LIN {X 0,Y 251.586,Z 580.66,A -85,B 0,C 180,E1 17106.896,E2 17106.896} C_VEL
LIN {X 0,Y 250.824,Z 580.66,A -85,B 0,C 180,E1 17115.723,E2 17115.723} C_VEL
LIN {X 0,Y 250.856,Z 581.328,A -85,B 0,C 180,E1 17116.877,E2 17116.877} C_VEL
LIN {X 0,Y 252.882,Z 586.254,A -85,B 0,C 180,E1 17118.487,E2 17118.487} C_VEL
LIN {X 0,Y 255.97,Z 589.116,A -85,B 0,C 180,E1 17120.381,E2 17120.381} C_VEL
LIN {X 0,Y 260.025,Z 594.777,A -85,B 0,C 180,E1 17122.728,E2 17122.728} C_VEL
LIN {X 0,Y 273.524,Z 615.35,A -85,B 0,C 180,E1 17129.206,E2 17129.206} C_VEL
LIN {X 0,Y 285.886,Z 637.872,A -85,B 0,C 180,E1 17134.459,E2 17134.459} C_VEL
LIN {X 0,Y 296.581,Z 664.88,A -85,B 0,C 180,E1 17139.344,E2 17139.344} C_VEL
LIN {X 0,Y 300.476,Z 680.869,A -85,B 0,C 180,E1 17141.812,E2 17141.812} C_VEL
LIN {X 0,Y 290.892,Z 714.694,A -85,B 0,C 180,E1 17144.762,E2 17144.762} C_VEL
LIN {X 0,Y 280.033,Z 747.013,A -85,B 0,C 180,E1 17149.078,E2 17149.078} C_VEL
LIN {X 0,Y 269.468,Z 775.475,A -85,B 0,C 180,E1 17154.67,E2 17154.67} C_VEL
LIN {X 0,Y 261.005,Z 799.602,A -85,B 0,C 180,E1 17161.584,E2 17161.584} C_VEL
LIN {X 0,Y 255.731,Z 817.938,A -85,B 0,C 180,E1 17169.263,E2 17169.263} C_VEL
LIN {X 0,Y 254.018,Z 830.311,A -85,B 0,C 180,E1 17177.144,E2 17177.144} C_VEL
LIN {X 0,Y 254.336,Z 835.933,A -85,B 0,C 180,E1 17183.183,E2 17183.183} C_VEL
LIN {X 0,Y 254.787,Z 838.259,A -85,B 0,C 180,E1 17189.997,E2 17189.997} C_VEL
LIN {X 0,Y 254.301,Z 835.944,A -85,B 0,C 180,E1 17196.813,E2 17196.813} C_VEL
LIN {X 0,Y 254.151,Z 828.084,A -85,B 0,C 180,E1 17204.612,E2 17204.612} C_VEL
LIN {X 0,Y 256.598,Z 814.491,A -85,B 0,C 180,E1 17212.469,E2 17212.469} C_VEL
LIN {X 0,Y 262.523,Z 794.979,A -85,B 0,C 180,E1 17219.974,E2 17219.974} C_VEL
LIN {X 0,Y 271.462,Z 770.337,A -85,B 0,C 180,E1 17226.54,E2 17226.54} C_VEL
LIN {X 0,Y 281.993,Z 741.378,A -85,B 0,C 180,E1 17231.838,E2 17231.838} C_VEL
LIN {X 0,Y 292.893,Z 708.642,A -85,B 0,C 180,E1 17235.888,E2 17235.888} C_VEL
LIN {X 0,Y 300.451,Z 679.152,A -85,B 0,C 180,E1 17238.429,E2 17238.429} C_VEL
LIN {X 0,Y 291.372,Z 650.188,A -85,B 0,C 180,E1 17243.212,E2 17243.212} C_VEL
LIN {X 0,Y 279.017,Z 624.432,A -85,B 0,C 180,E1 17248.514,E2 17248.514} C_VEL
LIN {X 0,Y 264.583,Z 601.351,A -85,B 0,C 180,E1 17255.009,E2 17255.009} C_VEL
LIN {X 0,Y 258.73,Z 593.721,A -85,B 0,C 180,E1 17258.055,E2 17258.055} C_VEL
LIN {X 0,Y 254.701,Z 587.628,A -85,B 0,C 180,E1 17260.528,E2 17260.528} C_VEL
LIN {X 0,Y 251.195,Z 583.366,A -85,B 0,C 180,E1 17262.902,E2 17262.902} C_VEL
LIN {X 0,Y 250.74,Z 580.66,A -85,B 0,C 180,E1 17263.513,E2 17263.513} C_VEL
LIN {X 0,Y 250.771,Z 580.66,A -85,B 0,C 180,E1 17264.591,E2 17264.591} C_VEL
LIN {X 0,Y 248.407,Z 580.66,A -85,B 0,C 180,E1 17267.555,E2 17267.555} C_VEL
LIN {X 0,Y 243.524,Z 580.66,A -85,B 0,C 180,E1 17272.588,E2 17272.588} C_VEL
LIN {X 0,Y 244.313,Z 580.66,A -85,B 0,C 180,E1 17279.993,E2 17279.993} C_VEL
LIN {X 0,Y 243.604,Z 580.66,A -85,B 0,C 180,E1 17287.689,E2 17287.689} C_VEL
LIN {X 0,Y 242.887,Z 581.231,A -85,B 0,C 180,E1 17296.498,E2 17296.498} C_VEL
LIN {X 0,Y 245.095,Z 586.44,A -85,B 0,C 180,E1 17299.111,E2 17299.111} C_VEL
LIN {X 0,Y 248.217,Z 589.119,A -85,B 0,C 180,E1 17301.735,E2 17301.735} C_VEL
LIN {X 0,Y 251.98,Z 594.885,A -85,B 0,C 180,E1 17304.775,E2 17304.775} C_VEL
LIN {X 0,Y 258.821,Z 606.093,A -85,B 0,C 180,E1 17309.635,E2 17309.635} C_VEL
LIN {X 0,Y 266.343,Z 619.396,A -85,B 0,C 180,E1 17314.5,E2 17314.5} C_VEL
LIN {X 0,Y 275.183,Z 640.528,A -85,B 0,C 180,E1 17320.618,E2 17320.618} C_VEL
LIN {X 0,Y 280.604,Z 660.927,A -85,B 0,C 180,E1 17325.778,E2 17325.778} C_VEL
LIN {X 0,Y 283.15,Z 682.748,A -85,B 0,C 180,E1 17331.089,E2 17331.089} C_VEL
LIN {X 0,Y 282.39,Z 690.579,A -85,B 0,C 180,E1 17332.879,E2 17332.879} C_VEL
LIN {X 0,Y 271.737,Z 715.104,A -85,B 0,C 180,E1 17338.165,E2 17338.165} C_VEL
LIN {X 0,Y 262.088,Z 734.388,A -85,B 0,C 180,E1 17344.421,E2 17344.421} C_VEL
LIN {X 0,Y 254.304,Z 749.195,A -85,B 0,C 180,E1 17351.948,E2 17351.948} C_VEL
LIN {X 0,Y 249.965,Z 757.81,A -85,B 0,C 180,E1 17359.569,E2 17359.569} C_VEL
LIN {X 0,Y 248.341,Z 761.384,A -85,B 0,C 180,E1 17366.52,E2 17366.52} C_VEL
LIN {X 0,Y 248.401,Z 761.339,A -85,B 0,C 180,E1 17373.486,E2 17373.486} C_VEL
LIN {X 0,Y 250.691,Z 756.218,A -85,B 0,C 180,E1 17382.164,E2 17382.164} C_VEL
LIN {X 0,Y 256.072,Z 745.785,A -85,B 0,C 180,E1 17390.024,E2 17390.024} C_VEL
LIN {X 0,Y 264.332,Z 729.864,A -85,B 0,C 180,E1 17397.176,E2 17397.176} C_VEL
LIN {X 0,Y 274.613,Z 708.641,A -85,B 0,C 180,E1 17403.334,E2 17403.334} C_VEL
LIN {X 0,Y 283.087,Z 687.119,A -85,B 0,C 180,E1 17407.736,E2 17407.736} C_VEL
LIN {X 0,Y 281.313,Z 665.464,A -85,B 0,C 180,E1 17413.014,E2 17413.014} C_VEL
LIN {X 0,Y 276.056,Z 643.398,A -85,B 0,C 180,E1 17418.477,E2 17418.477} C_VEL
LIN {X 0,Y 268.072,Z 623.359,A -85,B 0,C 180,E1 17424.148,E2 17424.148} C_VEL
LIN {X 0,Y 259.698,Z 607.475,A -85,B 0,C 180,E1 17429.607,E2 17429.607} C_VEL
LIN {X 0,Y 251.831,Z 594.8,A -85,B 0,C 180,E1 17435.08,E2 17435.08} C_VEL
LIN {X 0,Y 248.171,Z 589.103,A -85,B 0,C 180,E1 17438.026,E2 17438.026} C_VEL
LIN {X 0,Y 243.16,Z 583.155,A -85,B 0,C 180,E1 17442.656,E2 17442.656} C_VEL
LIN {X 0,Y 242.76,Z 580.66,A -85,B 0,C 180,E1 17443.348,E2 17443.348} C_VEL
LIN {X 0,Y 243.579,Z 580.66,A -85,B 0,C 180,E1 17452.89,E2 17452.89} C_VEL
LIN {X 0,Y 244.286,Z 580.66,A -85,B 0,C 180,E1 17460.007,E2 17460.007} C_VEL
LIN {X 0,Y 243.579,Z 580.66,A -85,B 0,C 180,E1 17467.599,E2 17467.599} C_VEL
LIN {X 0,Y 243.293,Z 581.322,A -85,B 0,C 180,E1 17471.182,E2 17471.182} C_VEL
LIN {X 0,Y 245.218,Z 586.034,A -85,B 0,C 180,E1 17473.348,E2 17473.348} C_VEL
LIN {X 0,Y 248.738,Z 589.237,A -85,B 0,C 180,E1 17476.195,E2 17476.195} C_VEL
LIN {X 0,Y 252.376,Z 594.794,A -85,B 0,C 180,E1 17478.864,E2 17478.864} C_VEL
LIN {X 0,Y 259.902,Z 605.854,A -85,B 0,C 180,E1 17483.417,E2 17483.417} C_VEL
LIN {X 0,Y 270.347,Z 622.266,A -85,B 0,C 180,E1 17488.668,E2 17488.668} C_VEL
LIN {X 0,Y 281.614,Z 643.967,A -85,B 0,C 180,E1 17493.894,E2 17493.894} C_VEL
LIN {X 0,Y 291.407,Z 670.701,A -85,B 0,C 180,E1 17498.927,E2 17498.927} C_VEL
LIN {X 0,Y 293.962,Z 683.793,A -85,B 0,C 180,E1 17500.965,E2 17500.965} C_VEL
LIN {X 0,Y 283.468,Z 718.719,A -85,B 0,C 180,E1 17504.224,E2 17504.224} C_VEL
LIN {X 0,Y 272.472,Z 749.515,A -85,B 0,C 180,E1 17508.614,E2 17508.614} C_VEL
LIN {X 0,Y 261.648,Z 777.115,A -85,B 0,C 180,E1 17514.349,E2 17514.349} C_VEL
LIN {X 0,Y 253.011,Z 800.517,A -85,B 0,C 180,E1 17521.5,E2 17521.5} C_VEL
LIN {X 0,Y 247.643,Z 818.557,A -85,B 0,C 180,E1 17529.58,E2 17529.58} C_VEL
LIN {X 0,Y 246.171,Z 829.932,A -85,B 0,C 180,E1 17537.467,E2 17537.467} C_VEL
LIN {X 0,Y 246.479,Z 834.73,A -85,B 0,C 180,E1 17542.964,E2 17542.964} C_VEL
LIN {X 0,Y 246.965,Z 837.071,A -85,B 0,C 180,E1 17549.997,E2 17549.997} C_VEL
LIN {X 0,Y 246.446,Z 834.741,A -85,B 0,C 180,E1 17557.031,E2 17557.031} C_VEL
LIN {X 0,Y 246.335,Z 826.853,A -85,B 0,C 180,E1 17565.087,E2 17565.087} C_VEL
LIN {X 0,Y 249.016,Z 813.226,A -85,B 0,C 180,E1 17573.192,E2 17573.192} C_VEL
LIN {X 0,Y 255.521,Z 793.456,A -85,B 0,C 180,E1 17580.975,E2 17580.975} C_VEL
LIN {X 0,Y 265.153,Z 768.4,A -85,B 0,C 180,E1 17587.736,E2 17587.736} C_VEL
LIN {X 0,Y 276.224,Z 739.373,A -85,B 0,C 180,E1 17593.062,E2 17593.062} C_VEL
LIN {X 0,Y 287.3,Z 707.205,A -85,B 0,C 180,E1 17597.048,E2 17597.048} C_VEL
LIN {X 0,Y 294.084,Z 681.567,A -85,B 0,C 180,E1 17599.32,E2 17599.32} C_VEL
LIN {X 0,Y 285.773,Z 653.755,A -85,B 0,C 180,E1 17604.182,E2 17604.182} C_VEL
LIN {X 0,Y 274.795,Z 629.935,A -85,B 0,C 180,E1 17609.355,E2 17609.355} C_VEL
LIN {X 0,Y 261.915,Z 608.278,A -85,B 0,C 180,E1 17615.646,E2 17615.646} C_VEL
LIN {X 0,Y 252.419,Z 594.824,A -85,B 0,C 180,E1 17621.252,E2 17621.252} C_VEL
LIN {X 0,Y 248.765,Z 589.298,A -85,B 0,C 180,E1 17623.95,E2 17623.95} C_VEL
LIN {X 0,Y 243.476,Z 582.895,A -85,B 0,C 180,E1 17628.714,E2 17628.714} C_VEL
LIN {X 0,Y 243.245,Z 580.66,A -85,B 0,C 180,E1 17629.268,E2 17629.268} C_VEL
LIN {X 0,Y 243.524,Z 580.66,A -85,B 0,C 180,E1 17632.588,E2 17632.588} C_VEL
LIN {X 0,Y 241.56,Z 580.866,A -85,B 0,C 180,E1 17635.609,E2 17635.609} C_VEL
LIN {X 0,Y 236.308,Z 581.372,A -85,B 0,C 180,E1 17640.735,E2 17640.735} C_VEL
LIN {X 0,Y 236.125,Z 582.654,A -85,B 0,C 180,E1 17645.034,E2 17645.034} C_VEL
LIN {X 0,Y 241.213,Z 589.227,A -85,B 0,C 180,E1 17655.935,E2 17655.935} C_VEL
LIN {X 0,Y 244.265,Z 594.75,A -85,B 0,C 180,E1 17659.521,E2 17659.521} C_VEL
LIN {X 0,Y 246.174,Z 596.995,A -85,B 0,C 180,E1 17661.317,E2 17661.317} C_VEL
LIN {X 0,Y 251.017,Z 604.941,A -85,B 0,C 180,E1 17665.534,E2 17665.534} C_VEL
LIN {X 0,Y 257.986,Z 617.049,A -85,B 0,C 180,E1 17670.773,E2 17670.773} C_VEL
LIN {X 0,Y 266.924,Z 636.801,A -85,B 0,C 180,E1 17677.416,E2 17677.416} C_VEL
LIN {X 0,Y 273.626,Z 659.052,A -85,B 0,C 180,E1 17683.579,E2 17683.579} C_VEL
LIN {X 0,Y 276.511,Z 682.15,A -85,B 0,C 180,E1 17689.455,E2 17689.455} C_VEL
LIN {X 0,Y 276.319,Z 691.581,A -85,B 0,C 180,E1 17691.853,E2 17691.853} C_VEL
LIN {X 0,Y 265.14,Z 716.323,A -85,B 0,C 180,E1 17697.276,E2 17697.276} C_VEL
LIN {X 0,Y 255.049,Z 735.593,A -85,B 0,C 180,E1 17703.662,E2 17703.662} C_VEL
LIN {X 0,Y 246.833,Z 750.462,A -85,B 0,C 180,E1 17711.439,E2 17711.439} C_VEL
LIN {X 0,Y 242.281,Z 758.998,A -85,B 0,C 180,E1 17719.235,E2 17719.235} C_VEL
LIN {X 0,Y 240.563,Z 762.567,A -85,B 0,C 180,E1 17726.407,E2 17726.407} C_VEL
LIN {X 0,Y 240.61,Z 762.525,A -85,B 0,C 180,E1 17733.599,E2 17733.599} C_VEL
LIN {X 0,Y 242.41,Z 758.874,A -85,B 0,C 180,E1 17740.766,E2 17740.766} C_VEL
LIN {X 0,Y 247.584,Z 749.058,A -85,B 0,C 180,E1 17749.377,E2 17749.377} C_VEL
LIN {X 0,Y 256.295,Z 733.262,A -85,B 0,C 180,E1 17757.15,E2 17757.15} C_VEL
LIN {X 0,Y 266.64,Z 712.908,A -85,B 0,C 180,E1 17763.491,E2 17763.491} C_VEL
LIN {X 0,Y 276.473,Z 689.578,A -85,B 0,C 180,E1 17768.516,E2 17768.516} C_VEL
LIN {X 0,Y 275.106,Z 668.329,A -85,B 0,C 180,E1 17773.924,E2 17773.924} C_VEL
LIN {X 0,Y 270.275,Z 646.652,A -85,B 0,C 180,E1 17779.593,E2 17779.593} C_VEL
LIN {X 0,Y 262.338,Z 625.74,A -85,B 0,C 180,E1 17785.898,E2 17785.898} C_VEL
LIN {X 0,Y 253.002,Z 608.092,A -85,B 0,C 180,E1 17792.719,E2 17792.719} C_VEL
LIN {X 0,Y 248.7,Z 601.295,A -85,B 0,C 180,E1 17796.152,E2 17796.152} C_VEL
LIN {X 0,Y 244.968,Z 595.242,A -85,B 0,C 180,E1 17799.546,E2 17799.546} C_VEL
LIN {X 0,Y 241.374,Z 590.26,A -85,B 0,C 180,E1 17803.368,E2 17803.368} C_VEL
LIN {X 0,Y 240.62,Z 588.252,A -85,B 0,C 180,E1 17804.452,E2 17804.452} C_VEL
LIN {X 0,Y 235.904,Z 581.705,A -85,B 0,C 180,E1 17815.076,E2 17815.076} C_VEL
LIN {X 0,Y 236.078,Z 580.66,A -85,B 0,C 180,E1 17816.342,E2 17816.342} C_VEL
LIN {X 0,Y 236.288,Z 581.54,A -85,B 0,C 180,E1 17820.693,E2 17820.693} C_VEL
LIN {X 0,Y 239.8,Z 587.635,A -85,B 0,C 180,E1 17828.388,E2 17828.388} C_VEL
LIN {X 0,Y 241.633,Z 589.26,A -85,B 0,C 180,E1 17830.576,E2 17830.576} C_VEL
LIN {X 0,Y 244.962,Z 594.756,A -85,B 0,C 180,E1 17834.043,E2 17834.043} C_VEL
LIN {X 0,Y 246.995,Z 597.157,A -85,B 0,C 180,E1 17835.735,E2 17835.735} C_VEL
LIN {X 0,Y 252.731,Z 605.965,A -85,B 0,C 180,E1 17839.97,E2 17839.97} C_VEL
LIN {X 0,Y 260.813,Z 618.329,A -85,B 0,C 180,E1 17844.805,E2 17844.805} C_VEL
LIN {X 0,Y 272.421,Z 639.11,A -85,B 0,C 180,E1 17850.826,E2 17850.826} C_VEL
LIN {X 0,Y 282.893,Z 665.351,A -85,B 0,C 180,E1 17856.451,E2 17856.451} C_VEL
LIN {X 0,Y 287.919,Z 685.239,A -85,B 0,C 180,E1 17859.975,E2 17859.975} C_VEL
LIN {X 0,Y 277.123,Z 719.417,A -85,B 0,C 180,E1 17863.279,E2 17863.279} C_VEL
LIN {X 0,Y 265.896,Z 749.338,A -85,B 0,C 180,E1 17867.649,E2 17867.649} C_VEL
LIN {X 0,Y 254.445,Z 777.14,A -85,B 0,C 180,E1 17873.625,E2 17873.625} C_VEL
LIN {X 0,Y 245.387,Z 800.43,A -85,B 0,C 180,E1 17881.034,E2 17881.034} C_VEL
LIN {X 0,Y 239.746,Z 818.454,A -85,B 0,C 180,E1 17889.597,E2 17889.597} C_VEL
LIN {X 0,Y 238.305,Z 828.85,A -85,B 0,C 180,E1 17897.193,E2 17897.193} C_VEL
LIN {X 0,Y 238.603,Z 833.523,A -85,B 0,C 180,E1 17902.731,E2 17902.731} C_VEL
LIN {X 0,Y 239.168,Z 835.886,A -85,B 0,C 180,E1 17909.997,E2 17909.997} C_VEL
LIN {X 0,Y 238.571,Z 833.536,A -85,B 0,C 180,E1 17917.264,E2 17917.264} C_VEL
LIN {X 0,Y 238.535,Z 825.622,A -85,B 0,C 180,E1 17925.592,E2 17925.592} C_VEL
LIN {X 0,Y 241.516,Z 811.968,A -85,B 0,C 180,E1 17933.957,E2 17933.957} C_VEL
LIN {X 0,Y 248.658,Z 791.721,A -85,B 0,C 180,E1 17942.106,E2 17942.106} C_VEL
LIN {X 0,Y 258.886,Z 766.728,A -85,B 0,C 180,E1 17948.921,E2 17948.921} C_VEL
LIN {X 0,Y 270.352,Z 738.015,A -85,B 0,C 180,E1 17954.236,E2 17954.236} C_VEL
LIN {X 0,Y 282.033,Z 705.186,A -85,B 0,C 180,E1 17958.307,E2 17958.307} C_VEL
LIN {X 0,Y 287.845,Z 684.025,A -85,B 0,C 180,E1 17960.236,E2 17960.236} C_VEL
LIN {X 0,Y 280.608,Z 658.457,A -85,B 0,C 180,E1 17964.931,E2 17964.931} C_VEL
LIN {X 0,Y 270.497,Z 635.303,A -85,B 0,C 180,E1 17970.205,E2 17970.205} C_VEL
LIN {X 0,Y 258.809,Z 614.731,A -85,B 0,C 180,E1 17976.478,E2 17976.478} C_VEL
LIN {X 0,Y 250.138,Z 601.941,A -85,B 0,C 180,E1 17981.985,E2 17981.985} C_VEL
LIN {X 0,Y 245.7,Z 595.309,A -85,B 0,C 180,E1 17985.546,E2 17985.546} C_VEL
LIN {X 0,Y 241.796,Z 590.037,A -85,B 0,C 180,E1 17989.431,E2 17989.431} C_VEL
LIN {X 0,Y 240.958,Z 588.207,A -85,B 0,C 180,E1 17990.532,E2 17990.532} C_VEL
LIN {X 0,Y 236.471,Z 582.27,A -85,B 0,C 180,E1 17999.422,E2 17999.422} C_VEL
LIN {X 0,Y 236.308,Z 581.372,A -85,B 0,C 180,E1 18000.735,E2 18000.735} C_VEL
LIN {X 0,Y 235.751,Z 584.741,A -85,B 0,C 180,E1 18003.811,E2 18003.811} C_VEL
LIN {X 0,Y 235.654,Z 592.641,A -85,B 0,C 180,E1 18008.292,E2 18008.292} C_VEL
LIN {X 0,Y 235.807,Z 593.017,A -85,B 0,C 180,E1 18008.823,E2 18008.823} C_VEL
LIN {X 0,Y 239.544,Z 597.051,A -85,B 0,C 180,E1 18015.512,E2 18015.512} C_VEL
LIN {X 0,Y 242.844,Z 602.654,A -85,B 0,C 180,E1 18019.64,E2 18019.64} C_VEL
LIN {X 0,Y 248.489,Z 612.571,A -85,B 0,C 180,E1 18025.257,E2 18025.257} C_VEL
LIN {X 0,Y 256.058,Z 626.846,A -85,B 0,C 180,E1 18031.524,E2 18031.524} C_VEL
LIN {X 0,Y 263.903,Z 647.737,A -85,B 0,C 180,E1 18038.419,E2 18038.419} C_VEL
LIN {X 0,Y 268.677,Z 668.607,A -85,B 0,C 180,E1 18044.28,E2 18044.28} C_VEL
LIN {X 0,Y 270.122,Z 690.297,A -85,B 0,C 180,E1 18050.079,E2 18050.079} C_VEL
LIN {X 0,Y 268.68,Z 696.548,A -85,B 0,C 180,E1 18051.516,E2 18051.516} C_VEL
LIN {X 0,Y 257.134,Z 720.302,A -85,B 0,C 180,E1 18057.128,E2 18057.128} C_VEL
LIN {X 0,Y 246.954,Z 738.807,A -85,B 0,C 180,E1 18063.709,E2 18063.709} C_VEL
LIN {X 0,Y 238.828,Z 752.674,A -85,B 0,C 180,E1 18071.588,E2 18071.588} C_VEL
LIN {X 0,Y 234.615,Z 760.184,A -85,B 0,C 180,E1 18078.879,E2 18078.879} C_VEL
LIN {X 0,Y 232.783,Z 763.751,A -85,B 0,C 180,E1 18086.287,E2 18086.287} C_VEL
LIN {X 0,Y 232.832,Z 763.709,A -85,B 0,C 180,E1 18093.719,E2 18093.719} C_VEL
LIN {X 0,Y 234.739,Z 760.062,A -85,B 0,C 180,E1 18101.122,E2 18101.122} C_VEL
LIN {X 0,Y 240.233,Z 750.217,A -85,B 0,C 180,E1 18110.021,E2 18110.021} C_VEL
LIN {X 0,Y 249.362,Z 734.467,A -85,B 0,C 180,E1 18117.97,E2 18117.97} C_VEL
LIN {X 0,Y 260.159,Z 714.146,A -85,B 0,C 180,E1 18124.44,E2 18124.44} C_VEL
LIN {X 0,Y 269.899,Z 692.288,A -85,B 0,C 180,E1 18129.259,E2 18129.259} C_VEL
LIN {X 0,Y 269.003,Z 671.834,A -85,B 0,C 180,E1 18134.719,E2 18134.719} C_VEL
LIN {X 0,Y 264.834,Z 650.819,A -85,B 0,C 180,E1 18140.507,E2 18140.507} C_VEL
LIN {X 0,Y 257.735,Z 630.957,A -85,B 0,C 180,E1 18146.819,E2 18146.819} C_VEL
LIN {X 0,Y 249.233,Z 614.042,A -85,B 0,C 180,E1 18153.811,E2 18153.811} C_VEL
LIN {X 0,Y 245.725,Z 607.992,A -85,B 0,C 180,E1 18156.987,E2 18156.987} C_VEL
LIN {X 0,Y 242.789,Z 602.637,A -85,B 0,C 180,E1 18160.097,E2 18160.097} C_VEL
LIN {X 0,Y 239.473,Z 597.266,A -85,B 0,C 180,E1 18164.117,E2 18164.117} C_VEL
LIN {X 0,Y 238.348,Z 595.598,A -85,B 0,C 180,E1 18165.807,E2 18165.807} C_VEL
LIN {X 0,Y 234.947,Z 588.74,A -85,B 0,C 180,E1 18175.979,E2 18175.979} C_VEL
LIN {X 0,Y 235.237,Z 589.167,A -85,B 0,C 180,E1 18180.237,E2 18180.237} C_VEL
LIN {X 0,Y 238.803,Z 595.516,A -85,B 0,C 180,E1 18188.409,E2 18188.409} C_VEL
LIN {X 0,Y 240.253,Z 597.512,A -85,B 0,C 180,E1 18190.295,E2 18190.295} C_VEL
LIN {X 0,Y 245.165,Z 604.866,A -85,B 0,C 180,E1 18195.284,E2 18195.284} C_VEL
LIN {X 0,Y 253.067,Z 616.91,A -85,B 0,C 180,E1 18201.197,E2 18201.197} C_VEL
LIN {X 0,Y 263.446,Z 635.507,A -85,B 0,C 180,E1 18207.508,E2 18207.508} C_VEL
LIN {X 0,Y 272.54,Z 655.544,A -85,B 0,C 180,E1 18212.676,E2 18212.676} C_VEL
LIN {X 0,Y 280.612,Z 681.66,A -85,B 0,C 180,E1 18217.995,E2 18217.995} C_VEL
LIN {X 0,Y 281.189,Z 689.045,A -85,B 0,C 180,E1 18219.152,E2 18219.152} C_VEL
LIN {X 0,Y 270.281,Z 721.706,A -85,B 0,C 180,E1 18222.485,E2 18222.485} C_VEL
LIN {X 0,Y 258.366,Z 751.708,A -85,B 0,C 180,E1 18227.11,E2 18227.11} C_VEL
LIN {X 0,Y 246.501,Z 778.966,A -85,B 0,C 180,E1 18233.353,E2 18233.353} C_VEL
LIN {X 0,Y 237.317,Z 801.448,A -85,B 0,C 180,E1 18240.996,E2 18240.996} C_VEL
LIN {X 0,Y 231.773,Z 818.528,A -85,B 0,C 180,E1 18249.731,E2 18249.731} C_VEL
LIN {X 0,Y 230.456,Z 829.476,A -85,B 0,C 180,E1 18258.669,E2 18258.669} C_VEL
LIN {X 0,Y 230.952,Z 834.022,A -85,B 0,C 180,E1 18266.251,E2 18266.251} C_VEL
LIN {X 0,Y 231.343,Z 834.698,A -85,B 0,C 180,E1 18269.997,E2 18269.997} C_VEL
LIN {X 0,Y 230.714,Z 832.332,A -85,B 0,C 180,E1 18277.513,E2 18277.513} C_VEL
LIN {X 0,Y 230.75,Z 824.39,A -85,B 0,C 180,E1 18286.133,E2 18286.133} C_VEL
LIN {X 0,Y 234.231,Z 810.115,A -85,B 0,C 180,E1 18295.064,E2 18295.064} C_VEL
LIN {X 0,Y 241.779,Z 790.207,A -85,B 0,C 180,E1 18303.228,E2 18303.228} C_VEL
LIN {X 0,Y 252.437,Z 765.642,A -85,B 0,C 180,E1 18310.042,E2 18310.042} C_VEL
LIN {X 0,Y 264.531,Z 736.646,A -85,B 0,C 180,E1 18315.477,E2 18315.477} C_VEL
LIN {X 0,Y 276.743,Z 703.54,A -85,B 0,C 180,E1 18319.579,E2 18319.579} C_VEL
LIN {X 0,Y 281.66,Z 686.633,A -85,B 0,C 180,E1 18321.145,E2 18321.145} C_VEL
LIN {X 0,Y 274.698,Z 661.035,A -85,B 0,C 180,E1 18326.158,E2 18326.158} C_VEL
LIN {X 0,Y 265.786,Z 639.989,A -85,B 0,C 180,E1 18331.257,E2 18331.257} C_VEL
LIN {X 0,Y 255.551,Z 621.092,A -85,B 0,C 180,E1 18337.31,E2 18337.31} C_VEL
LIN {X 0,Y 247.8,Z 608.961,A -85,B 0,C 180,E1 18342.725,E2 18342.725} C_VEL
LIN {X 0,Y 243.607,Z 602.49,A -85,B 0,C 180,E1 18346.334,E2 18346.334} C_VEL
LIN {X 0,Y 240.071,Z 596.887,A -85,B 0,C 180,E1 18350.269,E2 18350.269} C_VEL
LIN {X 0,Y 235.318,Z 589.217,A -85,B 0,C 180,E1 18360.912,E2 18360.912} C_VEL
LIN {X 0,Y 235.141,Z 590.695,A -85,B 0,C 180,E1 18365.286,E2 18365.286} C_VEL
LIN {X 0,Y 235.807,Z 593.017,A -85,B 0,C 180,E1 18368.823,E2 18368.823} C_VEL
LIN {X 0,Y 236.703,Z 597.349,A -85,B 0,C 180,E1 18371.829,E2 18371.829} C_VEL
LIN {X 0,Y 238.461,Z 607.278,A -85,B 0,C 180,E1 18376.624,E2 18376.624} C_VEL
LIN {X 0,Y 241.672,Z 612.262,A -85,B 0,C 180,E1 18380.589,E2 18380.589} C_VEL
LIN {X 0,Y 247.127,Z 622.339,A -85,B 0,C 180,E1 18386.266,E2 18386.266} C_VEL
LIN {X 0,Y 254.468,Z 639.652,A -85,B 0,C 180,E1 18393.293,E2 18393.293} C_VEL
LIN {X 0,Y 260.344,Z 658.969,A -85,B 0,C 180,E1 18399.599,E2 18399.599} C_VEL
LIN {X 0,Y 263.251,Z 678.268,A -85,B 0,C 180,E1 18405.13,E2 18405.13} C_VEL
LIN {X 0,Y 263.472,Z 695.175,A -85,B 0,C 180,E1 18409.887,E2 18409.887} C_VEL
LIN {X 0,Y 252.14,Z 718.764,A -85,B 0,C 180,E1 18415.356,E2 18415.356} C_VEL
LIN {X 0,Y 241.14,Z 737.999,A -85,B 0,C 180,E1 18422.014,E2 18422.014} C_VEL
LIN {X 0,Y 233.031,Z 751.329,A -85,B 0,C 180,E1 18429.14,E2 18429.14} C_VEL
LIN {X 0,Y 227.728,Z 759.927,A -85,B 0,C 180,E1 18436.594,E2 18436.594} C_VEL
LIN {X 0,Y 224.996,Z 764.937,A -85,B 0,C 180,E1 18446.158,E2 18446.158} C_VEL
LIN {X 0,Y 225.038,Z 764.896,A -85,B 0,C 180,E1 18453.848,E2 18453.848} C_VEL
LIN {X 0,Y 227.058,Z 761.253,A -85,B 0,C 180,E1 18461.503,E2 18461.503} C_VEL
LIN {X 0,Y 231.951,Z 752.892,A -85,B 0,C 180,E1 18469.628,E2 18469.628} C_VEL
LIN {X 0,Y 240.669,Z 738.716,A -85,B 0,C 180,E1 18477.545,E2 18477.545} C_VEL
LIN {X 0,Y 251.486,Z 719.753,A -85,B 0,C 180,E1 18484.232,E2 18484.232} C_VEL
LIN {X 0,Y 263.038,Z 696.595,A -85,B 0,C 180,E1 18489.651,E2 18489.651} C_VEL
LIN {X 0,Y 263.136,Z 677.702,A -85,B 0,C 180,E1 18494.893,E2 18494.893} C_VEL
LIN {X 0,Y 259.816,Z 656.967,A -85,B 0,C 180,E1 18500.843,E2 18500.843} C_VEL
LIN {X 0,Y 253.386,Z 636.621,A -85,B 0,C 180,E1 18507.601,E2 18507.601} C_VEL
LIN {X 0,Y 245.683,Z 620.028,A -85,B 0,C 180,E1 18514.806,E2 18514.806} C_VEL
LIN {X 0,Y 240.473,Z 610.042,A -85,B 0,C 180,E1 18520.516,E2 18520.516} C_VEL
LIN {X 0,Y 237.438,Z 604.196,A -85,B 0,C 180,E1 18524.884,E2 18524.884} C_VEL
LIN {X 0,Y 233.846,Z 596.301,A -85,B 0,C 180,E1 18537.233,E2 18537.233} C_VEL
LIN {X 0,Y 234.093,Z 597.56,A -85,B 0,C 180,E1 18540.353,E2 18540.353} C_VEL
LIN {X 0,Y 238.54,Z 604.82,A -85,B 0,C 180,E1 18549.679,E2 18549.679} C_VEL
LIN {X 0,Y 243.278,Z 612.629,A -85,B 0,C 180,E1 18554.945,E2 18554.945} C_VEL
LIN {X 0,Y 250.591,Z 624.544,A -85,B 0,C 180,E1 18560.839,E2 18560.839} C_VEL
LIN {X 0,Y 260.124,Z 642.708,A -85,B 0,C 180,E1 18567.175,E2 18567.175} C_VEL
LIN {X 0,Y 268.657,Z 663.487,A -85,B 0,C 180,E1 18572.592,E2 18572.592} C_VEL
LIN {X 0,Y 275.356,Z 688.69,A -85,B 0,C 180,E1 18577.855,E2 18577.855} C_VEL
LIN {X 0,Y 264.082,Z 722.391,A -85,B 0,C 180,E1 18581.45,E2 18581.45} C_VEL
LIN {X 0,Y 251.227,Z 753.016,A -85,B 0,C 180,E1 18586.36,E2 18586.36} C_VEL
LIN {X 0,Y 239.254,Z 779.231,A -85,B 0,C 180,E1 18592.622,E2 18592.622} C_VEL
LIN {X 0,Y 229.725,Z 801.258,A -85,B 0,C 180,E1 18600.483,E2 18600.483} C_VEL
LIN {X 0,Y 224.023,Z 817.708,A -85,B 0,C 180,E1 18609.288,E2 18609.288} C_VEL
LIN {X 0,Y 222.587,Z 828.253,A -85,B 0,C 180,E1 18618.263,E2 18618.263} C_VEL
LIN {X 0,Y 223.101,Z 832.827,A -85,B 0,C 180,E1 18626.119,E2 18626.119} C_VEL
LIN {X 0,Y 223.526,Z 833.51,A -85,B 0,C 180,E1 18629.997,E2 18629.997} C_VEL
LIN {X 0,Y 222.853,Z 831.127,A -85,B 0,C 180,E1 18637.779,E2 18637.779} C_VEL
LIN {X 0,Y 222.805,Z 824.282,A -85,B 0,C 180,E1 18645.714,E2 18645.714} C_VEL
LIN {X 0,Y 226.247,Z 810.524,A -85,B 0,C 180,E1 18655.077,E2 18655.077} C_VEL
LIN {X 0,Y 234.217,Z 790.509,A -85,B 0,C 180,E1 18663.772,E2 18663.772} C_VEL
LIN {X 0,Y 245.311,Z 766.319,A -85,B 0,C 180,E1 18670.806,E2 18670.806} C_VEL
LIN {X 0,Y 257.88,Z 737.687,A -85,B 0,C 180,E1 18676.389,E2 18676.389} C_VEL
LIN {X 0,Y 270.087,Z 706.326,A -85,B 0,C 180,E1 18680.439,E2 18680.439} C_VEL
LIN {X 0,Y 275.407,Z 688.869,A -85,B 0,C 180,E1 18682.158,E2 18682.158} C_VEL
LIN {X 0,Y 268.997,Z 664.167,A -85,B 0,C 180,E1 18687.284,E2 18687.284} C_VEL
LIN {X 0,Y 260.337,Z 642.985,A -85,B 0,C 180,E1 18692.8,E2 18692.8} C_VEL
LIN {X 0,Y 251.163,Z 625.571,A -85,B 0,C 180,E1 18698.865,E2 18698.865} C_VEL
LIN {X 0,Y 244.848,Z 615.359,A -85,B 0,C 180,E1 18703.779,E2 18703.779} C_VEL
LIN {X 0,Y 241.409,Z 609.673,A -85,B 0,C 180,E1 18707.128,E2 18707.128} C_VEL
LIN {X 0,Y 237.73,Z 603.421,A -85,B 0,C 180,E1 18711.783,E2 18711.783} C_VEL
LIN {X 0,Y 234.104,Z 597.034,A -85,B 0,C 180,E1 18721.84,E2 18721.84} C_VEL
LIN {X 0,Y 237.683,Z 604.673,A -85,B 0,C 180,E1 18735.091,E2 18735.091} C_VEL
LIN {X 0,Y 238.461,Z 607.278,A -85,B 0,C 180,E1 18736.624,E2 18736.624} C_VEL
LIN {X 0,Y 240.35,Z 615.537,A -85,B 0,C 180,E1 18740.278,E2 18740.278} C_VEL
LIN {X 0,Y 241.957,Z 625.473,A -85,B 0,C 180,E1 18743.764,E2 18743.764} C_VEL
LIN {X 0,Y 248.621,Z 641.235,A -85,B 0,C 180,E1 18751.049,E2 18751.049} C_VEL
LIN {X 0,Y 254.466,Z 661.408,A -85,B 0,C 180,E1 18758.142,E2 18758.142} C_VEL
LIN {X 0,Y 257.071,Z 680.392,A -85,B 0,C 180,E1 18763.92,E2 18763.92} C_VEL
LIN {X 0,Y 256.88,Z 698.408,A -85,B 0,C 180,E1 18769.197,E2 18769.197} C_VEL
LIN {X 0,Y 244.974,Z 721.36,A -85,B 0,C 180,E1 18774.732,E2 18774.732} C_VEL
LIN {X 0,Y 234.197,Z 739.308,A -85,B 0,C 180,E1 18781.163,E2 18781.163} C_VEL
LIN {X 0,Y 224.851,Z 753.828,A -85,B 0,C 180,E1 18789.375,E2 18789.375} C_VEL
LIN {X 0,Y 219.303,Z 762.559,A -85,B 0,C 180,E1 18798.091,E2 18798.091} C_VEL
LIN {X 0,Y 217.218,Z 766.12,A -85,B 0,C 180,E1 18806.02,E2 18806.02} C_VEL
LIN {X 0,Y 217.262,Z 766.08,A -85,B 0,C 180,E1 18813.986,E2 18813.986} C_VEL
LIN {X 0,Y 219.408,Z 762.442,A -85,B 0,C 180,E1 18821.91,E2 18821.91} C_VEL
LIN {X 0,Y 224.916,Z 753.653,A -85,B 0,C 180,E1 18830.626,E2 18830.626} C_VEL
LIN {X 0,Y 234.382,Z 738.908,A -85,B 0,C 180,E1 18838.875,E2 18838.875} C_VEL
LIN {X 0,Y 245.871,Z 719.597,A -85,B 0,C 180,E1 18845.667,E2 18845.667} C_VEL
LIN {X 0,Y 256.85,Z 697.924,A -85,B 0,C 180,E1 18850.805,E2 18850.805} C_VEL
LIN {X 0,Y 256.821,Z 677.546,A -85,B 0,C 180,E1 18856.787,E2 18856.787} C_VEL
LIN {X 0,Y 253.412,Z 657.239,A -85,B 0,C 180,E1 18863.047,E2 18863.047} C_VEL
LIN {X 0,Y 247.591,Z 638.704,A -85,B 0,C 180,E1 18869.823,E2 18869.823} C_VEL
LIN {X 0,Y 241.158,Z 623.505,A -85,B 0,C 180,E1 18876.988,E2 18876.988} C_VEL
LIN {X 0,Y 237.345,Z 616.698,A -85,B 0,C 180,E1 18881.722,E2 18881.722} C_VEL
LIN {X 0,Y 234.763,Z 610.907,A -85,B 0,C 180,E1 18886.297,E2 18886.297} C_VEL
LIN {X 0,Y 232.541,Z 604.091,A -85,B 0,C 180,E1 18897.26,E2 18897.26} C_VEL
LIN {X 0,Y 232.719,Z 605.251,A -85,B 0,C 180,E1 18900.007,E2 18900.007} C_VEL
LIN {X 0,Y 236.706,Z 612.498,A -85,B 0,C 180,E1 18909.292,E2 18909.292} C_VEL
LIN {X 0,Y 241.176,Z 620.332,A -85,B 0,C 180,E1 18914.615,E2 18914.615} C_VEL
LIN {X 0,Y 247.713,Z 631.583,A -85,B 0,C 180,E1 18920.327,E2 18920.327} C_VEL
LIN {X 0,Y 256.634,Z 649.807,A -85,B 0,C 180,E1 18926.847,E2 18926.847} C_VEL
LIN {X 0,Y 264.595,Z 671.54,A -85,B 0,C 180,E1 18932.584,E2 18932.584} C_VEL
LIN {X 0,Y 269.237,Z 691.261,A -85,B 0,C 180,E1 18936.86,E2 18936.86} C_VEL
LIN {X 0,Y 257.195,Z 724.805,A -85,B 0,C 180,E1 18940.618,E2 18940.618} C_VEL
LIN {X 0,Y 243.857,Z 754.857,A -85,B 0,C 180,E1 18945.669,E2 18945.669} C_VEL
LIN {X 0,Y 231.018,Z 781.619,A -85,B 0,C 180,E1 18952.535,E2 18952.535} C_VEL
LIN {X 0,Y 221.184,Z 803.203,A -85,B 0,C 180,E1 18960.914,E2 18960.914} C_VEL
LIN {X 0,Y 215.727,Z 819.214,A -85,B 0,C 180,E1 18970.529,E2 18970.529} C_VEL
LIN {X 0,Y 214.798,Z 828.377,A -85,B 0,C 180,E1 18979.599,E2 18979.599} C_VEL
LIN {X 0,Y 215.247,Z 831.63,A -85,B 0,C 180,E1 18985.977,E2 18985.977} C_VEL
LIN {X 0,Y 215.699,Z 832.321,A -85,B 0,C 180,E1 18989.997,E2 18989.997} C_VEL
LIN {X 0,Y 214.999,Z 829.923,A -85,B 0,C 180,E1 18998.066,E2 18998.066} C_VEL
LIN {X 0,Y 215.005,Z 823.048,A -85,B 0,C 180,E1 19006.3,E2 19006.3} C_VEL
LIN {X 0,Y 218.526,Z 810.125,A -85,B 0,C 180,E1 19015.485,E2 19015.485} C_VEL
LIN {X 0,Y 226.733,Z 790.688,A -85,B 0,C 180,E1 19024.399,E2 19024.399} C_VEL
LIN {X 0,Y 238.326,Z 766.725,A -85,B 0,C 180,E1 19031.662,E2 19031.662} C_VEL
LIN {X 0,Y 251.812,Z 737.528,A -85,B 0,C 180,E1 19037.539,E2 19037.539} C_VEL
LIN {X 0,Y 264.811,Z 705.368,A -85,B 0,C 180,E1 19041.741,E2 19041.741} C_VEL
LIN {X 0,Y 269.257,Z 691.595,A -85,B 0,C 180,E1 19043.138,E2 19043.138} C_VEL
LIN {X 0,Y 263.488,Z 667.778,A -85,B 0,C 180,E1 19048.361,E2 19048.361} C_VEL
LIN {X 0,Y 255.949,Z 648.303,A -85,B 0,C 180,E1 19053.721,E2 19053.721} C_VEL
LIN {X 0,Y 246.781,Z 629.639,A -85,B 0,C 180,E1 19060.575,E2 19060.575} C_VEL
LIN {X 0,Y 239.457,Z 617.19,A -85,B 0,C 180,E1 19067.483,E2 19067.483} C_VEL
LIN {X 0,Y 235.666,Z 610.817,A -85,B 0,C 180,E1 19072.636,E2 19072.636} C_VEL
LIN {X 0,Y 232.78,Z 604.823,A -85,B 0,C 180,E1 19081.85,E2 19081.85} C_VEL
LIN {X 0,Y 235.549,Z 612.254,A -85,B 0,C 180,E1 19094.691,E2 19094.691} C_VEL
LIN {X 0,Y 239.276,Z 620.225,A -85,B 0,C 180,E1 19100.541,E2 19100.541} C_VEL
LIN {X 0,Y 241.957,Z 625.473,A -85,B 0,C 180,E1 19103.764,E2 19103.764} C_VEL
LIN {X 0,Y 243.195,Z 636.122,A -85,B 0,C 180,E1 19107.057,E2 19107.057} C_VEL
LIN {X 0,Y 244.28,Z 647.028,A -85,B 0,C 180,E1 19110.32,E2 19110.32} C_VEL
LIN {X 0,Y 249.017,Z 665.878,A -85,B 0,C 180,E1 19117.287,E2 19117.287} C_VEL
LIN {X 0,Y 251.066,Z 684.784,A -85,B 0,C 180,E1 19123.329,E2 19123.329} C_VEL
LIN {X 0,Y 250.159,Z 701.521,A -85,B 0,C 180,E1 19128.436,E2 19128.436} C_VEL
LIN {X 0,Y 237.805,Z 723.962,A -85,B 0,C 180,E1 19134.064,E2 19134.064} C_VEL
LIN {X 0,Y 226.077,Z 742.509,A -85,B 0,C 180,E1 19141.127,E2 19141.127} C_VEL
LIN {X 0,Y 216.686,Z 756.249,A -85,B 0,C 180,E1 19149.628,E2 19149.628} C_VEL
LIN {X 0,Y 211.664,Z 763.745,A -85,B 0,C 180,E1 19157.655,E2 19157.655} C_VEL
LIN {X 0,Y 209.443,Z 767.304,A -85,B 0,C 180,E1 19165.872,E2 19165.872} C_VEL
LIN {X 0,Y 209.482,Z 767.265,A -85,B 0,C 180,E1 19174.134,E2 19174.134} C_VEL
LIN {X 0,Y 211.757,Z 763.633,A -85,B 0,C 180,E1 19182.347,E2 19182.347} C_VEL
LIN {X 0,Y 217.609,Z 754.846,A -85,B 0,C 180,E1 19191.352,E2 19191.352} C_VEL
LIN {X 0,Y 227.499,Z 740.204,A -85,B 0,C 180,E1 19199.787,E2 19199.787} C_VEL
LIN {X 0,Y 239.566,Z 720.821,A -85,B 0,C 180,E1 19206.756,E2 19206.756} C_VEL
LIN {X 0,Y 250.482,Z 699.865,A -85,B 0,C 180,E1 19211.895,E2 19211.895} C_VEL
LIN {X 0,Y 250.729,Z 679.326,A -85,B 0,C 180,E1 19218.216,E2 19218.216} C_VEL
LIN {X 0,Y 247.798,Z 660.406,A -85,B 0,C 180,E1 19224.441,E2 19224.441} C_VEL
LIN {X 0,Y 242.572,Z 642.504,A -85,B 0,C 180,E1 19231.47,E2 19231.47} C_VEL
LIN {X 0,Y 237.1,Z 629.053,A -85,B 0,C 180,E1 19238.543,E2 19238.543} C_VEL
LIN {X 0,Y 232.554,Z 618.417,A -85,B 0,C 180,E1 19246.736,E2 19246.736} C_VEL
LIN {X 0,Y 231.112,Z 611.814,A -85,B 0,C 180,E1 19258.221,E2 19258.221} C_VEL
LIN {X 0,Y 234.665,Z 620.094,A -85,B 0,C 180,E1 19268.907,E2 19268.907} C_VEL
LIN {X 0,Y 238.815,Z 627.886,A -85,B 0,C 180,E1 19274.295,E2 19274.295} C_VEL
LIN {X 0,Y 245.056,Z 639.66,A -85,B 0,C 180,E1 19280.256,E2 19280.256} C_VEL
LIN {X 0,Y 252.832,Z 656.737,A -85,B 0,C 180,E1 19286.458,E2 19286.458} C_VEL
LIN {X 0,Y 260.031,Z 678.995,A -85,B 0,C 180,E1 19292.469,E2 19292.469} C_VEL
LIN {X 0,Y 263.081,Z 694.838,A -85,B 0,C 180,E1 19296.009,E2 19296.009} C_VEL
LIN {X 0,Y 250.282,Z 727.348,A -85,B 0,C 180,E1 19299.76,E2 19299.76} C_VEL
LIN {X 0,Y 236.515,Z 756.659,A -85,B 0,C 180,E1 19304.956,E2 19304.956} C_VEL
LIN {X 0,Y 223.826,Z 781.732,A -85,B 0,C 180,E1 19311.716,E2 19311.716} C_VEL
LIN {X 0,Y 213.571,Z 802.977,A -85,B 0,C 180,E1 19320.355,E2 19320.355} C_VEL
LIN {X 0,Y 207.993,Z 818.134,A -85,B 0,C 180,E1 19329.913,E2 19329.913} C_VEL
LIN {X 0,Y 206.914,Z 827.157,A -85,B 0,C 180,E1 19339.198,E2 19339.198} C_VEL
LIN {X 0,Y 207.414,Z 830.437,A -85,B 0,C 180,E1 19345.825,E2 19345.825} C_VEL
LIN {X 0,Y 207.892,Z 831.135,A -85,B 0,C 180,E1 19349.996,E2 19349.996} C_VEL
LIN {X 0,Y 207.123,Z 828.714,A -85,B 0,C 180,E1 19358.374,E2 19358.374} C_VEL
LIN {X 0,Y 207.472,Z 820.585,A -85,B 0,C 180,E1 19368.095,E2 19368.095} C_VEL
LIN {X 0,Y 212.108,Z 806.145,A -85,B 0,C 180,E1 19377.991,E2 19377.991} C_VEL
LIN {X 0,Y 221.213,Z 786.957,A -85,B 0,C 180,E1 19386.519,E2 19386.519} C_VEL
LIN {X 0,Y 234.011,Z 761.905,A -85,B 0,C 180,E1 19393.877,E2 19393.877} C_VEL
LIN {X 0,Y 247.489,Z 733.782,A -85,B 0,C 180,E1 19399.31,E2 19399.31} C_VEL
LIN {X 0,Y 261.186,Z 700.577,A -85,B 0,C 180,E1 19403.474,E2 19403.474} C_VEL
LIN {X 0,Y 263.168,Z 694.557,A -85,B 0,C 180,E1 19404.079,E2 19404.079} C_VEL
LIN {X 0,Y 258.201,Z 672.003,A -85,B 0,C 180,E1 19409.293,E2 19409.293} C_VEL
LIN {X 0,Y 250.955,Z 652.081,A -85,B 0,C 180,E1 19415.103,E2 19415.103} C_VEL
LIN {X 0,Y 243.108,Z 635.644,A -85,B 0,C 180,E1 19421.633,E2 19421.633} C_VEL
LIN {X 0,Y 237.004,Z 624.448,A -85,B 0,C 180,E1 19428.052,E2 19428.052} C_VEL
LIN {X 0,Y 233.729,Z 618.365,A -85,B 0,C 180,E1 19433.041,E2 19433.041} C_VEL
LIN {X 0,Y 231.23,Z 612.57,A -85,B 0,C 180,E1 19441.863,E2 19441.863} C_VEL
LIN {X 0,Y 233.258,Z 619.734,A -85,B 0,C 180,E1 19454.31,E2 19454.31} C_VEL
LIN {X 0,Y 238.139,Z 630.501,A -85,B 0,C 180,E1 19462.336,E2 19462.336} C_VEL
LIN {X 0,Y 244.28,Z 647.028,A -85,B 0,C 180,E1 19470.32,E2 19470.32} C_VEL
LIN {X 0,Y 244.715,Z 655.377,A -85,B 0,C 180,E1 19472.693,E2 19472.693} C_VEL
LIN {X 0,Y 243.618,Z 670.583,A -85,B 0,C 180,E1 19476.486,E2 19476.486} C_VEL
LIN {X 0,Y 245.016,Z 688.82,A -85,B 0,C 180,E1 19482.632,E2 19482.632} C_VEL
LIN {X 0,Y 243.74,Z 704.013,A -85,B 0,C 180,E1 19487.494,E2 19487.494} C_VEL
LIN {X 0,Y 229.842,Z 727.893,A -85,B 0,C 180,E1 19493.786,E2 19493.786} C_VEL
LIN {X 0,Y 218.036,Z 745.417,A -85,B 0,C 180,E1 19501.028,E2 19501.028} C_VEL
LIN {X 0,Y 209.389,Z 757.438,A -85,B 0,C 180,E1 19508.884,E2 19508.884} C_VEL
LIN {X 0,Y 204.041,Z 764.932,A -85,B 0,C 180,E1 19517.186,E2 19517.186} C_VEL
LIN {X 0,Y 201.668,Z 768.488,A -85,B 0,C 180,E1 19525.713,E2 19525.713} C_VEL
LIN {X 0,Y 201.709,Z 768.449,A -85,B 0,C 180,E1 19534.294,E2 19534.294} C_VEL
LIN {X 0,Y 204.132,Z 764.82,A -85,B 0,C 180,E1 19542.816,E2 19542.816} C_VEL
LIN {X 0,Y 210.359,Z 756.036,A -85,B 0,C 180,E1 19552.126,E2 19552.126} C_VEL
LIN {X 0,Y 220.281,Z 742.119,A -85,B 0,C 180,E1 19560.469,E2 19560.469} C_VEL
LIN {X 0,Y 233.361,Z 722.044,A -85,B 0,C 180,E1 19567.903,E2 19567.903} C_VEL
LIN {X 0,Y 244.074,Z 702.371,A -85,B 0,C 180,E1 19572.851,E2 19572.851} C_VEL
LIN {X 0,Y 244.837,Z 684.04,A -85,B 0,C 180,E1 19578.772,E2 19578.772} C_VEL
LIN {X 0,Y 242.598,Z 665.048,A -85,B 0,C 180,E1 19585.374,E2 19585.374} C_VEL
LIN {X 0,Y 238.192,Z 647.859,A -85,B 0,C 180,E1 19592.491,E2 19592.491} C_VEL
LIN {X 0,Y 233.283,Z 634.341,A -85,B 0,C 180,E1 19600.157,E2 19600.157} C_VEL
LIN {X 0,Y 229.906,Z 625.629,A -85,B 0,C 180,E1 19607.618,E2 19607.618} C_VEL
LIN {X 0,Y 229.304,Z 619.537,A -85,B 0,C 180,E1 19618.506,E2 19618.506} C_VEL
LIN {X 0,Y 232.472,Z 627.723,A -85,B 0,C 180,E1 19628.621,E2 19628.621} C_VEL
LIN {X 0,Y 236.401,Z 635.681,A -85,B 0,C 180,E1 19634.209,E2 19634.209} C_VEL
LIN {X 0,Y 242.736,Z 648.404,A -85,B 0,C 180,E1 19640.649,E2 19640.649} C_VEL
LIN {X 0,Y 250.657,Z 668.901,A -85,B 0,C 180,E1 19647.746,E2 19647.746} C_VEL
LIN {X 0,Y 256.059,Z 690.713,A -85,B 0,C 180,E1 19653.425,E2 19653.425} C_VEL
LIN {X 0,Y 256.731,Z 697.969,A -85,B 0,C 180,E1 19654.995,E2 19654.995} C_VEL
LIN {X 0,Y 242.844,Z 730.984,A -85,B 0,C 180,E1 19659.037,E2 19659.037} C_VEL
LIN {X 0,Y 229.155,Z 758.561,A -85,B 0,C 180,E1 19664.263,E2 19664.263} C_VEL
LIN {X 0,Y 215.54,Z 783.999,A -85,B 0,C 180,E1 19671.584,E2 19671.584} C_VEL
LIN {X 0,Y 205.623,Z 803.44,A -85,B 0,C 180,E1 19680.175,E2 19680.175} C_VEL
LIN {X 0,Y 200.057,Z 817.953,A -85,B 0,C 180,E1 19690.005,E2 19690.005} C_VEL
LIN {X 0,Y 199.108,Z 826.862,A -85,B 0,C 180,E1 19700.161,E2 19700.161} C_VEL
LIN {X 0,Y 199.552,Z 829.239,A -85,B 0,C 180,E1 19705.66,E2 19705.66} C_VEL
LIN {X 0,Y 200.061,Z 829.946,A -85,B 0,C 180,E1 19709.996,E2 19709.996} C_VEL
LIN {X 0,Y 199.245,Z 827.505,A -85,B 0,C 180,E1 19718.708,E2 19718.708} C_VEL
LIN {X 0,Y 199.784,Z 819.353,A -85,B 0,C 180,E1 19728.817,E2 19728.817} C_VEL
LIN {X 0,Y 204.586,Z 805.605,A -85,B 0,C 180,E1 19738.669,E2 19738.669} C_VEL
LIN {X 0,Y 214.099,Z 786.724,A -85,B 0,C 180,E1 19747.431,E2 19747.431} C_VEL
LIN {X 0,Y 227.227,Z 762.419,A -85,B 0,C 180,E1 19754.87,E2 19754.87} C_VEL
LIN {X 0,Y 241.712,Z 733.631,A -85,B 0,C 180,E1 19760.576,E2 19760.576} C_VEL
LIN {X 0,Y 255.461,Z 701.721,A -85,B 0,C 180,E1 19764.666,E2 19764.666} C_VEL
LIN {X 0,Y 257.002,Z 696.487,A -85,B 0,C 180,E1 19765.278,E2 19765.278} C_VEL
LIN {X 0,Y 252.196,Z 673.832,A -85,B 0,C 180,E1 19770.908,E2 19770.908} C_VEL
LIN {X 0,Y 244.937,Z 653.273,A -85,B 0,C 180,E1 19777.52,E2 19777.52} C_VEL
LIN {X 0,Y 237.487,Z 637.497,A -85,B 0,C 180,E1 19784.807,E2 19784.807} C_VEL
LIN {X 0,Y 233.941,Z 631.021,A -85,B 0,C 180,E1 19789.189,E2 19789.189} C_VEL
LIN {X 0,Y 231.451,Z 625.715,A -85,B 0,C 180,E1 19793.677,E2 19793.677} C_VEL
LIN {X 0,Y 229.307,Z 620.279,A -85,B 0,C 180,E1 19802.586,E2 19802.586} C_VEL
LIN {X 0,Y 230.799,Z 627.387,A -85,B 0,C 180,E1 19814.054,E2 19814.054} C_VEL
LIN {X 0,Y 234.703,Z 637.179,A -85,B 0,C 180,E1 19821.687,E2 19821.687} C_VEL
LIN {X 0,Y 240.157,Z 654.148,A -85,B 0,C 180,E1 19830.166,E2 19830.166} C_VEL
LIN {X 0,Y 243.618,Z 670.583,A -85,B 0,C 180,E1 19836.486,E2 19836.486} C_VEL
LIN {X 0,Y 242.772,Z 679.296,A -85,B 0,C 180,E1 19838.792,E2 19838.792} C_VEL
LIN {X 0,Y 238.818,Z 694.669,A -85,B 0,C 180,E1 19842.509,E2 19842.509} C_VEL
LIN {X 0,Y 237.68,Z 705.893,A -85,B 0,C 180,E1 19846.354,E2 19846.354} C_VEL
LIN {X 0,Y 223.594,Z 729.102,A -85,B 0,C 180,E1 19852.605,E2 19852.605} C_VEL
LIN {X 0,Y 211.229,Z 746.614,A -85,B 0,C 180,E1 19860.001,E2 19860.001} C_VEL
LIN {X 0,Y 202.103,Z 758.629,A -85,B 0,C 180,E1 19868.084,E2 19868.084} C_VEL
LIN {X 0,Y 196.405,Z 766.124,A -85,B 0,C 180,E1 19876.678,E2 19876.678} C_VEL
LIN {X 0,Y 193.874,Z 769.675,A -85,B 0,C 180,E1 19885.54,E2 19885.54} C_VEL
LIN {X 0,Y 193.915,Z 769.637,A -85,B 0,C 180,E1 19894.467,E2 19894.467} C_VEL
LIN {X 0,Y 196.519,Z 766.009,A -85,B 0,C 180,E1 19903.321,E2 19903.321} C_VEL
LIN {X 0,Y 203.122,Z 757.23,A -85,B 0,C 180,E1 19912.959,E2 19912.959} C_VEL
LIN {X 0,Y 213.49,Z 743.437,A -85,B 0,C 180,E1 19921.483,E2 19921.483} C_VEL
LIN {X 0,Y 226.353,Z 724.645,A -85,B 0,C 180,E1 19928.683,E2 19928.683} C_VEL
LIN {X 0,Y 237.663,Z 705.284,A -85,B 0,C 180,E1 19933.715,E2 19933.715} C_VEL
LIN {X 0,Y 238.92,Z 686.669,A -85,B 0,C 180,E1 19940.058,E2 19940.058} C_VEL
LIN {X 0,Y 237.276,Z 669.204,A -85,B 0,C 180,E1 19946.48,E2 19946.48} C_VEL
LIN {X 0,Y 233.948,Z 653.931,A -85,B 0,C 180,E1 19953.17,E2 19953.17} C_VEL
LIN {X 0,Y 229.905,Z 640.916,A -85,B 0,C 180,E1 19960.851,E2 19960.851} C_VEL
LIN {X 0,Y 227.791,Z 633.895,A -85,B 0,C 180,E1 19966.602,E2 19966.602} C_VEL
LIN {X 0,Y 227.157,Z 627.37,A -85,B 0,C 180,E1 19978.437,E2 19978.437} C_VEL
LIN {X 0,Y 229.986,Z 635.231,A -85,B 0,C 180,E1 19988.325,E2 19988.325} C_VEL
LIN {X 0,Y 235.024,Z 645.746,A -85,B 0,C 180,E1 19995.615,E2 19995.615} C_VEL
LIN {X 0,Y 241.807,Z 662.365,A -85,B 0,C 180,E1 20002.961,E2 20002.961} C_VEL
LIN {X 0,Y 247.337,Z 680.118,A -85,B 0,C 180,E1 20008.719,E2 20008.719} C_VEL
LIN {X 0,Y 250.9,Z 698.687,A -85,B 0,C 180,E1 20013.571,E2 20013.571} C_VEL
LIN {X 0,Y 236.9,Z 731.484,A -85,B 0,C 180,E1 20017.809,E2 20017.809} C_VEL
LIN {X 0,Y 221.522,Z 760.947,A -85,B 0,C 180,E1 20023.632,E2 20023.632} C_VEL
LIN {X 0,Y 207.647,Z 785.328,A -85,B 0,C 180,E1 20031.184,E2 20031.184} C_VEL
LIN {X 0,Y 196.857,Z 805.567,A -85,B 0,C 180,E1 20040.947,E2 20040.947} C_VEL
LIN {X 0,Y 191.772,Z 819.299,A -85,B 0,C 180,E1 20051.651,E2 20051.651} C_VEL
LIN {X 0,Y 191.356,Z 826.27,A -85,B 0,C 180,E1 20060.922,E2 20060.922} C_VEL
LIN {X 0,Y 192.239,Z 828.758,A -85,B 0,C 180,E1 20069.996,E2 20069.996} C_VEL
LIN {X 0,Y 191.343,Z 826.29,A -85,B 0,C 180,E1 20079.071,E2 20079.071} C_VEL
LIN {X 0,Y 192.053,Z 818.261,A -85,B 0,C 180,E1 20089.452,E2 20089.452} C_VEL
LIN {X 0,Y 197.425,Z 804.392,A -85,B 0,C 180,E1 20099.784,E2 20099.784} C_VEL
LIN {X 0,Y 207.623,Z 785.45,A -85,B 0,C 180,E1 20108.812,E2 20108.812} C_VEL
LIN {X 0,Y 221.525,Z 761.128,A -85,B 0,C 180,E1 20116.358,E2 20116.358} C_VEL
LIN {X 0,Y 236.418,Z 732.701,A -85,B 0,C 180,E1 20122.032,E2 20122.032} C_VEL
LIN {X 0,Y 250.867,Z 700.359,A -85,B 0,C 180,E1 20126.159,E2 20126.159} C_VEL
LIN {X 0,Y 247.871,Z 681.76,A -85,B 0,C 180,E1 20130.85,E2 20130.85} C_VEL
LIN {X 0,Y 241.811,Z 662.068,A -85,B 0,C 180,E1 20137.213,E2 20137.213} C_VEL
LIN {X 0,Y 235.258,Z 646.306,A -85,B 0,C 180,E1 20144.27,E2 20144.27} C_VEL
LIN {X 0,Y 229.539,Z 633.59,A -85,B 0,C 180,E1 20153.15,E2 20153.15} C_VEL
LIN {X 0,Y 227.152,Z 627.996,A -85,B 0,C 180,E1 20162.551,E2 20162.551} C_VEL
LIN {X 0,Y 227.994,Z 634.306,A -85,B 0,C 180,E1 20173.386,E2 20173.386} C_VEL
LIN {X 0,Y 231.42,Z 644.679,A -85,B 0,C 180,E1 20181.56,E2 20181.56} C_VEL
LIN {X 0,Y 235.599,Z 659.836,A -85,B 0,C 180,E1 20189.439,E2 20189.439} C_VEL
LIN {X 0,Y 238.495,Z 677.731,A -85,B 0,C 180,E1 20196.608,E2 20196.608} C_VEL
LIN {X 0,Y 238.818,Z 694.669,A -85,B 0,C 180,E1 20202.509,E2 20202.509} C_VEL
LIN {X 0,Y 236.647,Z 700.637,A -85,B 0,C 180,E1 20203.963,E2 20203.963} C_VEL
LIN {X 0,Y 229.692,Z 711.329,A -85,B 0,C 180,E1 20205.977,E2 20205.977} C_VEL
LIN {X 0,Y 215.677,Z 732.817,A -85,B 0,C 180,E1 20212.258,E2 20212.258} C_VEL
LIN {X 0,Y 203.102,Z 749.632,A -85,B 0,C 180,E1 20219.906,E2 20219.906} C_VEL
LIN {X 0,Y 192.939,Z 762.123,A -85,B 0,C 180,E1 20229.432,E2 20229.432} C_VEL
LIN {X 0,Y 187.042,Z 769.584,A -85,B 0,C 180,E1 20240.719,E2 20240.719} C_VEL
LIN {X 0,Y 185.417,Z 771.388,A -85,B 0,C 180,E1 20250.004,E2 20250.004} C_VEL
LIN {X 0,Y 187.127,Z 769.518,A -85,B 0,C 180,E1 20259.285,E2 20259.285} C_VEL
LIN {X 0,Y 192.331,Z 762.781,A -85,B 0,C 180,E1 20269.735,E2 20269.735} C_VEL
LIN {X 0,Y 201.834,Z 751.07,A -85,B 0,C 180,E1 20279.078,E2 20279.078} C_VEL
LIN {X 0,Y 214.876,Z 733.741,A -85,B 0,C 180,E1 20287.281,E2 20287.281} C_VEL
LIN {X 0,Y 229.103,Z 712.045,A -85,B 0,C 180,E1 20293.72,E2 20293.72} C_VEL
LIN {X 0,Y 231.597,Z 706.442,A -85,B 0,C 180,E1 20295.257,E2 20295.257} C_VEL
LIN {X 0,Y 233.083,Z 688.793,A -85,B 0,C 180,E1 20301.605,E2 20301.605} C_VEL
LIN {X 0,Y 231.686,Z 671.104,A -85,B 0,C 180,E1 20308.609,E2 20308.609} C_VEL
LIN {X 0,Y 228.821,Z 656.607,A -85,B 0,C 180,E1 20315.67,E2 20315.67} C_VEL
LIN {X 0,Y 226.302,Z 646.611,A -85,B 0,C 180,E1 20322.111,E2 20322.111} C_VEL
LIN {X 0,Y 224.457,Z 640.366,A -85,B 0,C 180,E1 20328.373,E2 20328.373} C_VEL
LIN {X 0,Y 224.285,Z 635.853,A -85,B 0,C 180,E1 20336.15,E2 20336.15} C_VEL
LIN {X 0,Y 224.702,Z 636.495,A -85,B 0,C 180,E1 20340.007,E2 20340.007} C_VEL
LIN {X 0,Y 227.113,Z 642.063,A -85,B 0,C 180,E1 20347.643,E2 20347.643} C_VEL
LIN {X 0,Y 232.153,Z 654.025,A -85,B 0,C 180,E1 20355.813,E2 20355.813} C_VEL
LIN {X 0,Y 237.586,Z 668.637,A -85,B 0,C 180,E1 20362.406,E2 20362.406} C_VEL
LIN {X 0,Y 242.689,Z 687.49,A -85,B 0,C 180,E1 20368.649,E2 20368.649} C_VEL
LIN {X 0,Y 244.759,Z 702.426,A -85,B 0,C 180,E1 20372.656,E2 20372.656} C_VEL
LIN {X 0,Y 229.822,Z 734.368,A -85,B 0,C 180,E1 20376.887,E2 20376.887} C_VEL
LIN {X 0,Y 213.943,Z 763.064,A -85,B 0,C 180,E1 20382.963,E2 20382.963} C_VEL
LIN {X 0,Y 199.762,Z 786.656,A -85,B 0,C 180,E1 20390.752,E2 20390.752} C_VEL
LIN {X 0,Y 189.413,Z 804.897,A -85,B 0,C 180,E1 20400.135,E2 20400.135} C_VEL
LIN {X 0,Y 184.07,Z 818.061,A -85,B 0,C 180,E1 20410.854,E2 20410.854} C_VEL
LIN {X 0,Y 183.49,Z 825.146,A -85,B 0,C 180,E1 20420.726,E2 20420.726} C_VEL
LIN {X 0,Y 184.403,Z 827.567,A -85,B 0,C 180,E1 20429.996,E2 20429.996} C_VEL
LIN {X 0,Y 183.477,Z 825.08,A -85,B 0,C 180,E1 20439.463,E2 20439.463} C_VEL
LIN {X 0,Y 184.37,Z 817.019,A -85,B 0,C 180,E1 20450.297,E2 20450.297} C_VEL
LIN {X 0,Y 190.358,Z 803.137,A -85,B 0,C 180,E1 20461.009,E2 20461.009} C_VEL
LIN {X 0,Y 201.232,Z 784.167,A -85,B 0,C 180,E1 20470.291,E2 20470.291} C_VEL
LIN {X 0,Y 215.947,Z 759.827,A -85,B 0,C 180,E1 20477.932,E2 20477.932} C_VEL
LIN {X 0,Y 231.659,Z 731.045,A -85,B 0,C 180,E1 20483.668,E2 20483.668} C_VEL
LIN {X 0,Y 244.921,Z 701.256,A -85,B 0,C 180,E1 20487.637,E2 20487.637} C_VEL
LIN {X 0,Y 241.245,Z 680.514,A -85,B 0,C 180,E1 20493.486,E2 20493.486} C_VEL
LIN {X 0,Y 235.487,Z 662.111,A -85,B 0,C 180,E1 20500.336,E2 20500.336} C_VEL
LIN {X 0,Y 230.073,Z 648.987,A -85,B 0,C 180,E1 20507.386,E2 20507.386} C_VEL
LIN {X 0,Y 226.71,Z 640.795,A -85,B 0,C 180,E1 20513.784,E2 20513.784} C_VEL
LIN {X 0,Y 224.87,Z 635.916,A -85,B 0,C 180,E1 20521.314,E2 20521.314} C_VEL
LIN {X 0,Y 224.724,Z 640.54,A -85,B 0,C 180,E1 20531.613,E2 20531.613} C_VEL
LIN {X 0,Y 226.982,Z 649.151,A -85,B 0,C 180,E1 20539.405,E2 20539.405} C_VEL
LIN {X 0,Y 229.997,Z 660.793,A -85,B 0,C 180,E1 20546.401,E2 20546.401} C_VEL
LIN {X 0,Y 232.563,Z 677.474,A -85,B 0,C 180,E1 20553.87,E2 20553.87} C_VEL
LIN {X 0,Y 233.019,Z 694.537,A -85,B 0,C 180,E1 20560.346,E2 20560.346} C_VEL
LIN {X 0,Y 231.395,Z 708.378,A -85,B 0,C 180,E1 20565.295,E2 20565.295} C_VEL
LIN {X 0,Y 229.692,Z 711.329,A -85,B 0,C 180,E1 20565.977,E2 20565.977} C_VEL
LIN {X 0,Y 219.772,Z 723.029,A -85,B 0,C 180,E1 20568.18,E2 20568.18} C_VEL
LIN {X 0,Y 210.806,Z 732.394,A -85,B 0,C 180,E1 20570.364,E2 20570.364} C_VEL
LIN {X 0,Y 209.877,Z 733.586,A -85,B 0,C 180,E1 20570.789,E2 20570.789} C_VEL
LIN {X 0,Y 196.363,Z 750.833,A -85,B 0,C 180,E1 20578.76,E2 20578.76} C_VEL
LIN {X 0,Y 186.219,Z 762.679,A -85,B 0,C 180,E1 20587.906,E2 20587.906} C_VEL
LIN {X 0,Y 180.136,Z 769.743,A -85,B 0,C 180,E1 20597.916,E2 20597.916} C_VEL
LIN {X 0,Y 178.323,Z 772.045,A -85,B 0,C 180,E1 20605.15,E2 20605.15} C_VEL
LIN {X 0,Y 178.363,Z 772.007,A -85,B 0,C 180,E1 20614.857,E2 20614.857} C_VEL
LIN {X 0,Y 181.32,Z 768.389,A -85,B 0,C 180,E1 20624.461,E2 20624.461} C_VEL
LIN {X 0,Y 188.825,Z 759.612,A -85,B 0,C 180,E1 20634.809,E2 20634.809} C_VEL
LIN {X 0,Y 201.34,Z 744.494,A -85,B 0,C 180,E1 20644.492,E2 20644.492} C_VEL
LIN {X 0,Y 216.327,Z 724.304,A -85,B 0,C 180,E1 20652.177,E2 20652.177} C_VEL
LIN {X 0,Y 225.309,Z 709.574,A -85,B 0,C 180,E1 20656.156,E2 20656.156} C_VEL
LIN {X 0,Y 227.312,Z 692.035,A -85,B 0,C 180,E1 20662.809,E2 20662.809} C_VEL
LIN {X 0,Y 226.637,Z 676.01,A -85,B 0,C 180,E1 20669.555,E2 20669.555} C_VEL
LIN {X 0,Y 224.51,Z 661.706,A -85,B 0,C 180,E1 20676.927,E2 20676.927} C_VEL
LIN {X 0,Y 222.244,Z 651.732,A -85,B 0,C 180,E1 20684.25,E2 20684.25} C_VEL
LIN {X 0,Y 221.178,Z 646.846,A -85,B 0,C 180,E1 20690.188,E2 20690.188} C_VEL
LIN {X 0,Y 221.626,Z 643.433,A -85,B 0,C 180,E1 20696.104,E2 20696.104} C_VEL
LIN {X 0,Y 222.092,Z 644.077,A -85,B 0,C 180,E1 20700.007,E2 20700.007} C_VEL
LIN {X 0,Y 224.323,Z 649.9,A -85,B 0,C 180,E1 20707.738,E2 20707.738} C_VEL
LIN {X 0,Y 228.593,Z 660.784,A -85,B 0,C 180,E1 20715.316,E2 20715.316} C_VEL
LIN {X 0,Y 233.567,Z 676.044,A -85,B 0,C 180,E1 20722.312,E2 20722.312} C_VEL
LIN {X 0,Y 237.653,Z 694.133,A -85,B 0,C 180,E1 20728.442,E2 20728.442} C_VEL
LIN {X 0,Y 238.74,Z 705.045,A -85,B 0,C 180,E1 20731.462,E2 20731.462} C_VEL
LIN {X 0,Y 222.646,Z 737.396,A -85,B 0,C 180,E1 20735.993,E2 20735.993} C_VEL
LIN {X 0,Y 206.092,Z 765.534,A -85,B 0,C 180,E1 20742.328,E2 20742.328} C_VEL
LIN {X 0,Y 191.152,Z 789.034,A -85,B 0,C 180,E1 20750.834,E2 20750.834} C_VEL
LIN {X 0,Y 180.655,Z 806.744,A -85,B 0,C 180,E1 20761.019,E2 20761.019} C_VEL
LIN {X 0,Y 175.819,Z 819.143,A -85,B 0,C 180,E1 20772.692,E2 20772.692} C_VEL
LIN {X 0,Y 175.602,Z 823.843,A -85,B 0,C 180,E1 20780.1,E2 20780.1} C_VEL
LIN {X 0,Y 176.59,Z 826.38,A -85,B 0,C 180,E1 20789.996,E2 20789.996} C_VEL
LIN {X 0,Y 175.596,Z 823.865,A -85,B 0,C 180,E1 20799.892,E2 20799.892} C_VEL
LIN {X 0,Y 176.761,Z 815.73,A -85,B 0,C 180,E1 20811.268,E2 20811.268} C_VEL
LIN {X 0,Y 183.363,Z 801.878,A -85,B 0,C 180,E1 20822.332,E2 20822.332} C_VEL
LIN {X 0,Y 195.037,Z 782.893,A -85,B 0,C 180,E1 20831.852,E2 20831.852} C_VEL
LIN {X 0,Y 210.136,Z 759.154,A -85,B 0,C 180,E1 20839.433,E2 20839.433} C_VEL
LIN {X 0,Y 226.511,Z 730.526,A -85,B 0,C 180,E1 20845.188,E2 20845.188} C_VEL
LIN {X 0,Y 238.94,Z 703.971,A -85,B 0,C 180,E1 20848.812,E2 20848.812} C_VEL
LIN {X 0,Y 235.866,Z 684.176,A -85,B 0,C 180,E1 20854.775,E2 20854.775} C_VEL
LIN {X 0,Y 230.664,Z 666.376,A -85,B 0,C 180,E1 20861.89,E2 20861.89} C_VEL
LIN {X 0,Y 225.868,Z 653.62,A -85,B 0,C 180,E1 20869.407,E2 20869.407} C_VEL
LIN {X 0,Y 223.829,Z 648.025,A -85,B 0,C 180,E1 20874.189,E2 20874.189} C_VEL
LIN {X 0,Y 222.236,Z 644.481,A -85,B 0,C 180,E1 20879.993,E2 20879.993} C_VEL
LIN {X 0,Y 221.732,Z 643.969,A -85,B 0,C 180,E1 20883.895,E2 20883.895} C_VEL
LIN {X 0,Y 221.921,Z 648.977,A -85,B 0,C 180,E1 20892.734,E2 20892.734} C_VEL
LIN {X 0,Y 223.926,Z 658.282,A -85,B 0,C 180,E1 20900.71,E2 20900.71} C_VEL
LIN {X 0,Y 226.301,Z 671.932,A -85,B 0,C 180,E1 20908.392,E2 20908.392} C_VEL
LIN {X 0,Y 227.439,Z 688.193,A -85,B 0,C 180,E1 20915.508,E2 20915.508} C_VEL
LIN {X 0,Y 226.13,Z 705.614,A -85,B 0,C 180,E1 20922.199,E2 20922.199} C_VEL
LIN {X 0,Y 224.133,Z 712.598,A -85,B 0,C 180,E1 20924.6,E2 20924.6} C_VEL
LIN {X 0,Y 209.877,Z 733.586,A -85,B 0,C 180,E1 20930.789,E2 20930.789} C_VEL
LIN {X 0,Y 205.459,Z 738.444,A -85,B 0,C 180,E1 20932.394,E2 20932.394} C_VEL
LIN {X 0,Y 190.945,Z 750.649,A -85,B 0,C 180,E1 20936.752,E2 20936.752} C_VEL
LIN {X 0,Y 190.077,Z 751.597,A -85,B 0,C 180,E1 20937.281,E2 20937.281} C_VEL
LIN {X 0,Y 178.402,Z 764.472,A -85,B 0,C 180,E1 20947.633,E2 20947.633} C_VEL
LIN {X 0,Y 171.651,Z 771.954,A -85,B 0,C 180,E1 20959.878,E2 20959.878} C_VEL
LIN {X 0,Y 169.822,Z 773.757,A -85,B 0,C 180,E1 20970.004,E2 20970.004} C_VEL
LIN {X 0,Y 171.731,Z 771.89,A -85,B 0,C 180,E1 20980.125,E2 20980.125} C_VEL
LIN {X 0,Y 178.267,Z 764.542,A -85,B 0,C 180,E1 20992.132,E2 20992.132} C_VEL
LIN {X 0,Y 189.812,Z 751.79,A -85,B 0,C 180,E1 21002.456,E2 21002.456} C_VEL
LIN {X 0,Y 204.643,Z 733.651,A -85,B 0,C 180,E1 21010.878,E2 21010.878} C_VEL
LIN {X 0,Y 219.063,Z 712.634,A -85,B 0,C 180,E1 21017.137,E2 21017.137} C_VEL
LIN {X 0,Y 221.569,Z 694.965,A -85,B 0,C 180,E1 21024.213,E2 21024.213} C_VEL
LIN {X 0,Y 221.425,Z 678.783,A -85,B 0,C 180,E1 21031.519,E2 21031.519} C_VEL
LIN {X 0,Y 219.898,Z 665.868,A -85,B 0,C 180,E1 21038.893,E2 21038.893} C_VEL
LIN {X 0,Y 218.448,Z 656.405,A -85,B 0,C 180,E1 21046.934,E2 21046.934} C_VEL
LIN {X 0,Y 218.709,Z 650.935,A -85,B 0,C 180,E1 21056.051,E2 21056.051} C_VEL
LIN {X 0,Y 219.367,Z 652.976,A -85,B 0,C 180,E1 21061.978,E2 21061.978} C_VEL
LIN {X 0,Y 221.301,Z 657.615,A -85,B 0,C 180,E1 21067.845,E2 21067.845} C_VEL
LIN {X 0,Y 225.232,Z 668.654,A -85,B 0,C 180,E1 21075.551,E2 21075.551} C_VEL
LIN {X 0,Y 229.602,Z 684.559,A -85,B 0,C 180,E1 21082.719,E2 21082.719} C_VEL
LIN {X 0,Y 232.586,Z 702.532,A -85,B 0,C 180,E1 21088.802,E2 21088.802} C_VEL
LIN {X 0,Y 232.569,Z 708.049,A -85,B 0,C 180,E1 21090.267,E2 21090.267} C_VEL
LIN {X 0,Y 216.071,Z 739.348,A -85,B 0,C 180,E1 21094.854,E2 21094.854} C_VEL
LIN {X 0,Y 198.765,Z 767.062,A -85,B 0,C 180,E1 21101.434,E2 21101.434} C_VEL
LIN {X 0,Y 183.895,Z 789.196,A -85,B 0,C 180,E1 21109.903,E2 21109.903} C_VEL
LIN {X 0,Y 172.637,Z 807.088,A -85,B 0,C 180,E1 21120.947,E2 21120.947} C_VEL
LIN {X 0,Y 168.065,Z 818.039,A -85,B 0,C 180,E1 21132.051,E2 21132.051} C_VEL
LIN {X 0,Y 167.731,Z 823.502,A -85,B 0,C 180,E1 21141.769,E2 21141.769} C_VEL
LIN {X 0,Y 168.748,Z 825.189,A -85,B 0,C 180,E1 21149.996,E2 21149.996} C_VEL
LIN {X 0,Y 167.715,Z 822.649,A -85,B 0,C 180,E1 21160.362,E2 21160.362} C_VEL
LIN {X 0,Y 169.169,Z 814.488,A -85,B 0,C 180,E1 21172.272,E2 21172.272} C_VEL
LIN {X 0,Y 176.458,Z 800.615,A -85,B 0,C 180,E1 21183.762,E2 21183.762} C_VEL
LIN {X 0,Y 189.394,Z 781.068,A -85,B 0,C 180,E1 21193.739,E2 21193.739} C_VEL
LIN {X 0,Y 206.065,Z 756.03,A -85,B 0,C 180,E1 21201.615,E2 21201.615} C_VEL
LIN {X 0,Y 222.354,Z 728.486,A -85,B 0,C 180,E1 21207.018,E2 21207.018} C_VEL
LIN {X 0,Y 233.084,Z 706.894,A -85,B 0,C 180,E1 21209.967,E2 21209.967} C_VEL
LIN {X 0,Y 230.526,Z 688.232,A -85,B 0,C 180,E1 21215.949,E2 21215.949} C_VEL
LIN {X 0,Y 226.122,Z 671.222,A -85,B 0,C 180,E1 21223.235,E2 21223.235} C_VEL
LIN {X 0,Y 222.288,Z 660.111,A -85,B 0,C 180,E1 21230.222,E2 21230.222} C_VEL
LIN {X 0,Y 220.093,Z 654.434,A -85,B 0,C 180,E1 21236.062,E2 21236.062} C_VEL
LIN {X 0,Y 219.336,Z 651.924,A -85,B 0,C 180,E1 21239.993,E2 21239.993} C_VEL
LIN {X 0,Y 218.827,Z 651.426,A -85,B 0,C 180,E1 21243.946,E2 21243.946} C_VEL
LIN {X 0,Y 218.644,Z 656.725,A -85,B 0,C 180,E1 21253.054,E2 21253.054} C_VEL
LIN {X 0,Y 220.075,Z 666.188,A -85,B 0,C 180,E1 21261.089,E2 21261.089} C_VEL
LIN {X 0,Y 221.545,Z 679.146,A -85,B 0,C 180,E1 21268.465,E2 21268.465} C_VEL
LIN {X 0,Y 221.729,Z 694.113,A -85,B 0,C 180,E1 21275.257,E2 21275.257} C_VEL
LIN {X 0,Y 219.719,Z 710.005,A -85,B 0,C 180,E1 21281.689,E2 21281.689} C_VEL
LIN {X 0,Y 218.044,Z 714.873,A -85,B 0,C 180,E1 21283.403,E2 21283.403} C_VEL
LIN {X 0,Y 202.581,Z 736.496,A -85,B 0,C 180,E1 21290.032,E2 21290.032} C_VEL
LIN {X 0,Y 190.077,Z 751.597,A -85,B 0,C 180,E1 21297.281,E2 21297.281} C_VEL
LIN {X 0,Y 180.764,Z 758.981,A -85,B 0,C 180,E1 21301.275,E2 21301.275} C_VEL
LIN {X 0,Y 171.93,Z 764.946,A -85,B 0,C 180,E1 21305.814,E2 21305.814} C_VEL
LIN {X 0,Y 164.879,Z 772.116,A -85,B 0,C 180,E1 21316.779,E2 21316.779} C_VEL
LIN {X 0,Y 162.77,Z 774.416,A -85,B 0,C 180,E1 21324.685,E2 21324.685} C_VEL
LIN {X 0,Y 162.812,Z 774.379,A -85,B 0,C 180,E1 21335.322,E2 21335.322} C_VEL
LIN {X 0,Y 167.258,Z 769.665,A -85,B 0,C 180,E1 21347.845,E2 21347.845} C_VEL
LIN {X 0,Y 177.355,Z 759.272,A -85,B 0,C 180,E1 21359.293,E2 21359.293} C_VEL
LIN {X 0,Y 191.958,Z 743.18,A -85,B 0,C 180,E1 21368.97,E2 21368.97} C_VEL
LIN {X 0,Y 208.328,Z 722.192,A -85,B 0,C 180,E1 21376.416,E2 21376.416} C_VEL
LIN {X 0,Y 212.718,Z 715.81,A -85,B 0,C 180,E1 21378.096,E2 21378.096} C_VEL
LIN {X 0,Y 215.81,Z 699.826,A -85,B 0,C 180,E1 21384.847,E2 21384.847} C_VEL
LIN {X 0,Y 216.395,Z 685.223,A -85,B 0,C 180,E1 21391.743,E2 21391.743} C_VEL
LIN {X 0,Y 215.684,Z 672.095,A -85,B 0,C 180,E1 21399.534,E2 21399.534} C_VEL
LIN {X 0,Y 214.858,Z 663.891,A -85,B 0,C 180,E1 21406.711,E2 21406.711} C_VEL
LIN {X 0,Y 215.479,Z 658.318,A -85,B 0,C 180,E1 21415.992,E2 21415.992} C_VEL
LIN {X 0,Y 216.192,Z 660.293,A -85,B 0,C 180,E1 21422.007,E2 21422.007} C_VEL
LIN {X 0,Y 218,Z 665.138,A -85,B 0,C 180,E1 21427.964,E2 21427.964} C_VEL
LIN {X 0,Y 221.54,Z 676.551,A -85,B 0,C 180,E1 21435.817,E2 21435.817} C_VEL
LIN {X 0,Y 225.284,Z 693.002,A -85,B 0,C 180,E1 21443.179,E2 21443.179} C_VEL
LIN {X 0,Y 226.987,Z 709.377,A -85,B 0,C 180,E1 21448.743,E2 21448.743} C_VEL
LIN {X 0,Y 210.216,Z 740.201,A -85,B 0,C 180,E1 21453.437,E2 21453.437} C_VEL
LIN {X 0,Y 192.339,Z 767.328,A -85,B 0,C 180,E1 21460.097,E2 21460.097} C_VEL
LIN {X 0,Y 176.263,Z 789.915,A -85,B 0,C 180,E1 21469.164,E2 21469.164} C_VEL
LIN {X 0,Y 164.517,Z 807.532,A -85,B 0,C 180,E1 21481.045,E2 21481.045} C_VEL
LIN {X 0,Y 159.957,Z 818.429,A -85,B 0,C 180,E1 21493.556,E2 21493.556} C_VEL
LIN {X 0,Y 160.194,Z 823.237,A -85,B 0,C 180,E1 21504.591,E2 21504.591} C_VEL
LIN {X 0,Y 160.902,Z 823.997,A -85,B 0,C 180,E1 21509.995,E2 21509.995} C_VEL
LIN {X 0,Y 159.834,Z 821.432,A -85,B 0,C 180,E1 21520.879,E2 21520.879} C_VEL
LIN {X 0,Y 161.651,Z 813.248,A -85,B 0,C 180,E1 21533.368,E2 21533.368} C_VEL
LIN {X 0,Y 169.676,Z 799.356,A -85,B 0,C 180,E1 21545.307,E2 21545.307} C_VEL
LIN {X 0,Y 183.216,Z 780.269,A -85,B 0,C 180,E1 21555.314,E2 21555.314} C_VEL
LIN {X 0,Y 200.336,Z 755.904,A -85,B 0,C 180,E1 21563.157,E2 21563.157} C_VEL
LIN {X 0,Y 218.053,Z 727.147,A -85,B 0,C 180,E1 21568.802,E2 21568.802} C_VEL
LIN {X 0,Y 227.133,Z 709.209,A -85,B 0,C 180,E1 21571.346,E2 21571.346} C_VEL
LIN {X 0,Y 225.168,Z 691.87,A -85,B 0,C 180,E1 21577.329,E2 21577.329} C_VEL
LIN {X 0,Y 221.672,Z 676.786,A -85,B 0,C 180,E1 21584.193,E2 21584.193} C_VEL
LIN {X 0,Y 218.15,Z 665.426,A -85,B 0,C 180,E1 21592.041,E2 21592.041} C_VEL
LIN {X 0,Y 216.161,Z 659.257,A -85,B 0,C 180,E1 21599.993,E2 21599.993} C_VEL
LIN {X 0,Y 215.596,Z 658.767,A -85,B 0,C 180,E1 21604.006,E2 21604.006} C_VEL
LIN {X 0,Y 215.048,Z 664.19,A -85,B 0,C 180,E1 21613.277,E2 21613.277} C_VEL
LIN {X 0,Y 215.978,Z 673.479,A -85,B 0,C 180,E1 21621.24,E2 21621.24} C_VEL
LIN {X 0,Y 216.538,Z 685.817,A -85,B 0,C 180,E1 21628.369,E2 21628.369} C_VEL
LIN {X 0,Y 215.726,Z 701.642,A -85,B 0,C 180,E1 21635.792,E2 21635.792} C_VEL
LIN {X 0,Y 212.676,Z 716.196,A -85,B 0,C 180,E1 21641.889,E2 21641.889} C_VEL
LIN {X 0,Y 196.676,Z 737.704,A -85,B 0,C 180,E1 21648.574,E2 21648.574} C_VEL
LIN {X 0,Y 181.587,Z 754.876,A -85,B 0,C 180,E1 21657.313,E2 21657.313} C_VEL
LIN {X 0,Y 171.93,Z 764.946,A -85,B 0,C 180,E1 21665.814,E2 21665.814} C_VEL
LIN {X 0,Y 163.983,Z 769.83,A -85,B 0,C 180,E1 21670.892,E2 21670.892} C_VEL
LIN {X 0,Y 157.135,Z 773.444,A -85,B 0,C 180,E1 21676.511,E2 21676.511} C_VEL
LIN {X 0,Y 155.01,Z 775.6,A -85,B 0,C 180,E1 21684.419,E2 21684.419} C_VEL
LIN {X 0,Y 155.053,Z 775.563,A -85,B 0,C 180,E1 21695.589,E2 21695.589} C_VEL
LIN {X 0,Y 160.086,Z 770.588,A -85,B 0,C 180,E1 21709.144,E2 21709.144} C_VEL
LIN {X 0,Y 170.562,Z 760.467,A -85,B 0,C 180,E1 21720.581,E2 21720.581} C_VEL
LIN {X 0,Y 185.943,Z 744.392,A -85,B 0,C 180,E1 21730.486,E2 21730.486} C_VEL
LIN {X 0,Y 203.3,Z 723.084,A -85,B 0,C 180,E1 21738.1,E2 21738.1} C_VEL
LIN {X 0,Y 207.078,Z 717.185,A -85,B 0,C 180,E1 21739.862,E2 21739.862} C_VEL
LIN {X 0,Y 210.399,Z 701.667,A -85,B 0,C 180,E1 21746.869,E2 21746.869} C_VEL
LIN {X 0,Y 211.379,Z 688.644,A -85,B 0,C 180,E1 21753.513,E2 21753.513} C_VEL
LIN {X 0,Y 211.254,Z 676.437,A -85,B 0,C 180,E1 21761.507,E2 21761.507} C_VEL
LIN {X 0,Y 211.156,Z 668.845,A -85,B 0,C 180,E1 21769.488,E2 21769.488} C_VEL
LIN {X 0,Y 212.033,Z 665.583,A -85,B 0,C 180,E1 21775.927,E2 21775.927} C_VEL
LIN {X 0,Y 212.642,Z 666.142,A -85,B 0,C 180,E1 21780.008,E2 21780.008} C_VEL
LIN {X 0,Y 214.458,Z 672.502,A -85,B 0,C 180,E1 21788.097,E2 21788.097} C_VEL
LIN {X 0,Y 217.155,Z 682.551,A -85,B 0,C 180,E1 21795.111,E2 21795.111} C_VEL
LIN {X 0,Y 219.98,Z 697.528,A -85,B 0,C 180,E1 21802.171,E2 21802.171} C_VEL
LIN {X 0,Y 221.177,Z 712.362,A -85,B 0,C 180,E1 21807.508,E2 21807.508} C_VEL
LIN {X 0,Y 203.177,Z 742.933,A -85,B 0,C 180,E1 21812.345,E2 21812.345} C_VEL
LIN {X 0,Y 184.923,Z 769.152,A -85,B 0,C 180,E1 21819.173,E2 21819.173} C_VEL
LIN {X 0,Y 168.337,Z 790.91,A -85,B 0,C 180,E1 21828.613,E2 21828.613} C_VEL
LIN {X 0,Y 157.307,Z 806.396,A -85,B 0,C 180,E1 21839.705,E2 21839.705} C_VEL
LIN {X 0,Y 152.193,Z 817.194,A -85,B 0,C 180,E1 21852.691,E2 21852.691} C_VEL
LIN {X 0,Y 152.304,Z 822.033,A -85,B 0,C 180,E1 21864.309,E2 21864.309} C_VEL
LIN {X 0,Y 153.053,Z 822.805,A -85,B 0,C 180,E1 21869.995,E2 21869.995} C_VEL
LIN {X 0,Y 151.938,Z 820.21,A -85,B 0,C 180,E1 21881.452,E2 21881.452} C_VEL
LIN {X 0,Y 154.2,Z 812.01,A -85,B 0,C 180,E1 21894.57,E2 21894.57} C_VEL
LIN {X 0,Y 163.064,Z 798.102,A -85,B 0,C 180,E1 21906.97,E2 21906.97} C_VEL
LIN {X 0,Y 177.31,Z 779.278,A -85,B 0,C 180,E1 21917.083,E2 21917.083} C_VEL
LIN {X 0,Y 195.382,Z 754.844,A -85,B 0,C 180,E1 21925.016,E2 21925.016} C_VEL
LIN {X 0,Y 213.297,Z 726.953,A -85,B 0,C 180,E1 21930.484,E2 21930.484} C_VEL
LIN {X 0,Y 221.24,Z 712.749,A -85,B 0,C 180,E1 21932.446,E2 21932.446} C_VEL
LIN {X 0,Y 219.909,Z 696.466,A -85,B 0,C 180,E1 21938.351,E2 21938.351} C_VEL
LIN {X 0,Y 217.281,Z 682.774,A -85,B 0,C 180,E1 21944.899,E2 21944.899} C_VEL
LIN {X 0,Y 214.276,Z 671.643,A -85,B 0,C 180,E1 21952.957,E2 21952.957} C_VEL
LIN {X 0,Y 212.775,Z 666.484,A -85,B 0,C 180,E1 21959.992,E2 21959.992} C_VEL
LIN {X 0,Y 211.954,Z 666.299,A -85,B 0,C 180,E1 21964.718,E2 21964.718} C_VEL
LIN {X 0,Y 211.273,Z 670.463,A -85,B 0,C 180,E1 21972.364,E2 21972.364} C_VEL
LIN {X 0,Y 211.441,Z 678.472,A -85,B 0,C 180,E1 21979.795,E2 21979.795} C_VEL
LIN {X 0,Y 211.45,Z 689.99,A -85,B 0,C 180,E1 21987.05,E2 21987.05} C_VEL
LIN {X 0,Y 210.071,Z 704.46,A -85,B 0,C 180,E1 21994.276,E2 21994.276} C_VEL
LIN {X 0,Y 206.808,Z 718.497,A -85,B 0,C 180,E1 22000.559,E2 22000.559} C_VEL
LIN {X 0,Y 189.852,Z 740.134,A -85,B 0,C 180,E1 22007.507,E2 22007.507} C_VEL
LIN {X 0,Y 175.057,Z 756.069,A -85,B 0,C 180,E1 22015.93,E2 22015.93} C_VEL
LIN {X 0,Y 162.959,Z 767.905,A -85,B 0,C 180,E1 22026.831,E2 22026.831} C_VEL
LIN {X 0,Y 157.135,Z 773.444,A -85,B 0,C 180,E1 22036.511,E2 22036.511} C_VEL
LIN {X 0,Y 153.077,Z 775.383,A -85,B 0,C 180,E1 22041.084,E2 22041.084} C_VEL
LIN {X 0,Y 146.584,Z 777.211,A -85,B 0,C 180,E1 22048.262,E2 22048.262} C_VEL
LIN {X 0,Y 146.443,Z 777.234,A -85,B 0,C 180,E1 22049.123,E2 22049.123} C_VEL
LIN {X 0,Y 148.718,Z 775.449,A -85,B 0,C 180,E1 22061.713,E2 22061.713} C_VEL
LIN {X 0,Y 155.837,Z 768.964,A -85,B 0,C 180,E1 22074.305,E2 22074.305} C_VEL
LIN {X 0,Y 168.71,Z 757.056,A -85,B 0,C 180,E1 22085.551,E2 22085.551} C_VEL
LIN {X 0,Y 185.346,Z 739.814,A -85,B 0,C 180,E1 22094.607,E2 22094.607} C_VEL
LIN {X 0,Y 200.725,Z 720.933,A -85,B 0,C 180,E1 22100.705,E2 22100.705} C_VEL
LIN {X 0,Y 204.576,Z 706.503,A -85,B 0,C 180,E1 22107.532,E2 22107.532} C_VEL
LIN {X 0,Y 206.355,Z 692.512,A -85,B 0,C 180,E1 22115.146,E2 22115.146} C_VEL
LIN {X 0,Y 206.911,Z 681.552,A -85,B 0,C 180,E1 22123.049,E2 22123.049} C_VEL
LIN {X 0,Y 207.279,Z 675.823,A -85,B 0,C 180,E1 22129.523,E2 22129.523} C_VEL
LIN {X 0,Y 208.36,Z 672.762,A -85,B 0,C 180,E1 22135.855,E2 22135.855} C_VEL
LIN {X 0,Y 209.058,Z 673.276,A -85,B 0,C 180,E1 22140.008,E2 22140.008} C_VEL
LIN {X 0,Y 210.681,Z 679.782,A -85,B 0,C 180,E1 22148.243,E2 22148.243} C_VEL
LIN {X 0,Y 212.976,Z 690.242,A -85,B 0,C 180,E1 22155.415,E2 22155.415} C_VEL
LIN {X 0,Y 214.998,Z 705.446,A -85,B 0,C 180,E1 22162.557,E2 22162.557} C_VEL
LIN {X 0,Y 215.375,Z 714.548,A -85,B 0,C 180,E1 22165.976,E2 22165.976} C_VEL
LIN {X 0,Y 196.907,Z 744.632,A -85,B 0,C 180,E1 22170.977,E2 22170.977} C_VEL
LIN {X 0,Y 177.536,Z 770.78,A -85,B 0,C 180,E1 22178.164,E2 22178.164} C_VEL
LIN {X 0,Y 160.504,Z 791.78,A -85,B 0,C 180,E1 22187.94,E2 22187.94} C_VEL
LIN {X 0,Y 148.327,Z 808.072,A -85,B 0,C 180,E1 22201.099,E2 22201.099} C_VEL
LIN {X 0,Y 144.088,Z 817.567,A -85,B 0,C 180,E1 22214.818,E2 22214.818} C_VEL
LIN {X 0,Y 144.41,Z 820.827,A -85,B 0,C 180,E1 22223.997,E2 22223.997} C_VEL
LIN {X 0,Y 145.203,Z 821.612,A -85,B 0,C 180,E1 22229.995,E2 22229.995} C_VEL
LIN {X 0,Y 144.075,Z 818.99,A -85,B 0,C 180,E1 22242.086,E2 22242.086} C_VEL
LIN {X 0,Y 146.775,Z 810.763,A -85,B 0,C 180,E1 22255.902,E2 22255.902} C_VEL
LIN {X 0,Y 157.16,Z 796.127,A -85,B 0,C 180,E1 22269.271,E2 22269.271} C_VEL
LIN {X 0,Y 173.218,Z 776.288,A -85,B 0,C 180,E1 22279.822,E2 22279.822} C_VEL
LIN {X 0,Y 192.498,Z 751.026,A -85,B 0,C 180,E1 22287.655,E2 22287.655} C_VEL
LIN {X 0,Y 211.447,Z 722.225,A -85,B 0,C 180,E1 22292.93,E2 22292.93} C_VEL
LIN {X 0,Y 215.481,Z 714.686,A -85,B 0,C 180,E1 22294.038,E2 22294.038} C_VEL
LIN {X 0,Y 214.522,Z 699.832,A -85,B 0,C 180,E1 22299.939,E2 22299.939} C_VEL
LIN {X 0,Y 212.419,Z 686.996,A -85,B 0,C 180,E1 22306.645,E2 22306.645} C_VEL
LIN {X 0,Y 210.295,Z 677.774,A -85,B 0,C 180,E1 22313.902,E2 22313.902} C_VEL
LIN {X 0,Y 209.187,Z 673.589,A -85,B 0,C 180,E1 22319.992,E2 22319.992} C_VEL
LIN {X 0,Y 208.475,Z 673.12,A -85,B 0,C 180,E1 22324.143,E2 22324.143} C_VEL
LIN {X 0,Y 207.281,Z 677.686,A -85,B 0,C 180,E1 22332.606,E2 22332.606} C_VEL
LIN {X 0,Y 206.918,Z 685.586,A -85,B 0,C 180,E1 22340.004,E2 22340.004} C_VEL
LIN {X 0,Y 206.005,Z 697.779,A -85,B 0,C 180,E1 22347.691,E2 22347.691} C_VEL
LIN {X 0,Y 203.674,Z 711.591,A -85,B 0,C 180,E1 22354.795,E2 22354.795} C_VEL
LIN {X 0,Y 200.697,Z 721.287,A -85,B 0,C 180,E1 22359.272,E2 22359.272} C_VEL
LIN {X 0,Y 183.098,Z 742.475,A -85,B 0,C 180,E1 22366.361,E2 22366.361} C_VEL
LIN {X 0,Y 166.946,Z 758.885,A -85,B 0,C 180,E1 22375.61,E2 22375.61} C_VEL
LIN {X 0,Y 154.717,Z 770.054,A -85,B 0,C 180,E1 22387.044,E2 22387.044} C_VEL
LIN {X 0,Y 148.637,Z 775.511,A -85,B 0,C 180,E1 22398.291,E2 22398.291} C_VEL
LIN {X 0,Y 146.443,Z 777.234,A -85,B 0,C 180,E1 22409.123,E2 22409.123} C_VEL
LIN {X 0,Y 143.166,Z 777.581,A -85,B 0,C 180,E1 22415.937,E2 22415.937} C_VEL
LIN {X 0,Y 141.298,Z 776.419,A -85,B 0,C 180,E1 22422.985,E2 22422.985} C_VEL
LIN {X 0,Y 150.002,Z 769.095,A -85,B 0,C 180,E1 22436.921,E2 22436.921} C_VEL
LIN {X 0,Y 164.17,Z 756.688,A -85,B 0,C 180,E1 22448.268,E2 22448.268} C_VEL
LIN {X 0,Y 182.202,Z 738.5,A -85,B 0,C 180,E1 22457.312,E2 22457.312} C_VEL
LIN {X 0,Y 194.553,Z 723.964,A -85,B 0,C 180,E1 22461.976,E2 22461.976} C_VEL
LIN {X 0,Y 198.939,Z 710.587,A -85,B 0,C 180,E1 22468.609,E2 22468.609} C_VEL
LIN {X 0,Y 201.373,Z 697.24,A -85,B 0,C 180,E1 22476.34,E2 22476.34} C_VEL
LIN {X 0,Y 202.499,Z 687.279,A -85,B 0,C 180,E1 22484.051,E2 22484.051} C_VEL
LIN {X 0,Y 203.355,Z 681.719,A -85,B 0,C 180,E1 22491.474,E2 22491.474} C_VEL
LIN {X 0,Y 204.459,Z 679.805,A -85,B 0,C 180,E1 22495.776,E2 22495.776} C_VEL
LIN {X 0,Y 205.183,Z 680.257,A -85,B 0,C 180,E1 22500.008,E2 22500.008} C_VEL
LIN {X 0,Y 206.446,Z 685.818,A -85,B 0,C 180,E1 22507.356,E2 22507.356} C_VEL
LIN {X 0,Y 208.21,Z 695.947,A -85,B 0,C 180,E1 22514.701,E2 22514.701} C_VEL
LIN {X 0,Y 209.57,Z 710.508,A -85,B 0,C 180,E1 22521.82,E2 22521.82} C_VEL
LIN {X 0,Y 208.927,Z 718.84,A -85,B 0,C 180,E1 22524.847,E2 22524.847} C_VEL
LIN {X 0,Y 189.365,Z 748.092,A -85,B 0,C 180,E1 22529.932,E2 22529.932} C_VEL
LIN {X 0,Y 169.31,Z 773.415,A -85,B 0,C 180,E1 22537.466,E2 22537.466} C_VEL
LIN {X 0,Y 151.727,Z 793.712,A -85,B 0,C 180,E1 22547.994,E2 22547.994} C_VEL
LIN {X 0,Y 140.179,Z 808.275,A -85,B 0,C 180,E1 22561.189,E2 22561.189} C_VEL
LIN {X 0,Y 136.313,Z 816.34,A -85,B 0,C 180,E1 22573.929,E2 22573.929} C_VEL
LIN {X 0,Y 136.566,Z 819.706,A -85,B 0,C 180,E1 22584.031,E2 22584.031} C_VEL
LIN {X 0,Y 137.345,Z 820.419,A -85,B 0,C 180,E1 22589.995,E2 22589.995} C_VEL
LIN {X 0,Y 136.542,Z 819.641,A -85,B 0,C 180,E1 22596.339,E2 22596.339} C_VEL
LIN {X 0,Y 136.761,Z 814.768,A -85,B 0,C 180,E1 22609.324,E2 22609.324} C_VEL
LIN {X 0,Y 143.246,Z 804.002,A -85,B 0,C 180,E1 22623.568,E2 22623.568} C_VEL
LIN {X 0,Y 157.305,Z 787.432,A -85,B 0,C 180,E1 22636,E2 22636} C_VEL
LIN {X 0,Y 176.232,Z 765.205,A -85,B 0,C 180,E1 22645.49,E2 22645.49} C_VEL
LIN {X 0,Y 195.524,Z 739.732,A -85,B 0,C 180,E1 22651.856,E2 22651.856} C_VEL
LIN {X 0,Y 209.717,Z 717.149,A -85,B 0,C 180,E1 22655.572,E2 22655.572} C_VEL
LIN {X 0,Y 209.08,Z 702.161,A -85,B 0,C 180,E1 22662.054,E2 22662.054} C_VEL
LIN {X 0,Y 207.262,Z 689.807,A -85,B 0,C 180,E1 22669.506,E2 22669.506} C_VEL
LIN {X 0,Y 205.945,Z 683.158,A -85,B 0,C 180,E1 22675.791,E2 22675.791} C_VEL
LIN {X 0,Y 205.319,Z 680.554,A -85,B 0,C 180,E1 22679.992,E2 22679.992} C_VEL
LIN {X 0,Y 204.585,Z 680.131,A -85,B 0,C 180,E1 22684.222,E2 22684.222} C_VEL
LIN {X 0,Y 203.026,Z 684.766,A -85,B 0,C 180,E1 22692.875,E2 22692.875} C_VEL
LIN {X 0,Y 202.05,Z 693.004,A -85,B 0,C 180,E1 22700.508,E2 22700.508} C_VEL
LIN {X 0,Y 200.344,Z 704.802,A -85,B 0,C 180,E1 22708.054,E2 22708.054} C_VEL
LIN {X 0,Y 196.773,Z 718.694,A -85,B 0,C 180,E1 22715.377,E2 22715.377} C_VEL
LIN {X 0,Y 194.453,Z 724.312,A -85,B 0,C 180,E1 22717.982,E2 22717.982} C_VEL
LIN {X 0,Y 175.312,Z 745.96,A -85,B 0,C 180,E1 22725.633,E2 22725.633} C_VEL
LIN {X 0,Y 158.852,Z 761.614,A -85,B 0,C 180,E1 22735.26,E2 22735.26} C_VEL
LIN {X 0,Y 147.533,Z 771.244,A -85,B 0,C 180,E1 22745.857,E2 22745.857} C_VEL
LIN {X 0,Y 140.998,Z 776.696,A -85,B 0,C 180,E1 22757.646,E2 22757.646} C_VEL
LIN {X 0,Y 138.609,Z 778.498,A -85,B 0,C 180,E1 22770.005,E2 22770.005} C_VEL
LIN {X 0,Y 141.298,Z 776.419,A -85,B 0,C 180,E1 22782.985,E2 22782.985} C_VEL
LIN {X 0,Y 140.728,Z 774.4,A -85,B 0,C 180,E1 22790.067,E2 22790.067} C_VEL
LIN {X 0,Y 141.878,Z 771.231,A -85,B 0,C 180,E1 22797.062,E2 22797.062} C_VEL
LIN {X 0,Y 155.874,Z 759.756,A -85,B 0,C 180,E1 22808.664,E2 22808.664} C_VEL
LIN {X 0,Y 174.589,Z 742.241,A -85,B 0,C 180,E1 22818.202,E2 22818.202} C_VEL
LIN {X 0,Y 189.135,Z 725.867,A -85,B 0,C 180,E1 22823.728,E2 22823.728} C_VEL
LIN {X 0,Y 193.708,Z 713.135,A -85,B 0,C 180,E1 22830.548,E2 22830.548} C_VEL
LIN {X 0,Y 196.575,Z 700.661,A -85,B 0,C 180,E1 22838.494,E2 22838.494} C_VEL
LIN {X 0,Y 198.034,Z 692.992,A -85,B 0,C 180,E1 22845.088,E2 22845.088} C_VEL
LIN {X 0,Y 199.096,Z 688.592,A -85,B 0,C 180,E1 22851.29,E2 22851.29} C_VEL
LIN {X 0,Y 200.273,Z 686.665,A -85,B 0,C 180,E1 22855.687,E2 22855.687} C_VEL
LIN {X 0,Y 201.082,Z 687.101,A -85,B 0,C 180,E1 22860.008,E2 22860.008} C_VEL
LIN {X 0,Y 202.165,Z 692.835,A -85,B 0,C 180,E1 22867.513,E2 22867.513} C_VEL
LIN {X 0,Y 203.464,Z 703.374,A -85,B 0,C 180,E1 22875.054,E2 22875.054} C_VEL
LIN {X 0,Y 203.918,Z 718.707,A -85,B 0,C 180,E1 22882.469,E2 22882.469} C_VEL
LIN {X 0,Y 202.144,Z 722.986,A -85,B 0,C 180,E1 22883.534,E2 22883.534} C_VEL
LIN {X 0,Y 182.611,Z 750.478,A -85,B 0,C 180,E1 22888.596,E2 22888.596} C_VEL
LIN {X 0,Y 162.001,Z 774.848,A -85,B 0,C 180,E1 22896.299,E2 22896.299} C_VEL
LIN {X 0,Y 143.978,Z 794.354,A -85,B 0,C 180,E1 22907.204,E2 22907.204} C_VEL
LIN {X 0,Y 132.131,Z 808.339,A -85,B 0,C 180,E1 22921.159,E2 22921.159} C_VEL
LIN {X 0,Y 128.348,Z 816.514,A -85,B 0,C 180,E1 22936.395,E2 22936.395} C_VEL
LIN {X 0,Y 129.5,Z 819.227,A -85,B 0,C 180,E1 22949.994,E2 22949.994} C_VEL
LIN {X 0,Y 128.632,Z 818.432,A -85,B 0,C 180,E1 22956.731,E2 22956.731} C_VEL
LIN {X 0,Y 129.209,Z 813.343,A -85,B 0,C 180,E1 22970.864,E2 22970.864} C_VEL
LIN {X 0,Y 136.472,Z 802.751,A -85,B 0,C 180,E1 22985.477,E2 22985.477} C_VEL
LIN {X 0,Y 152.695,Z 785.071,A -85,B 0,C 180,E1 22998.887,E2 22998.887} C_VEL
LIN {X 0,Y 172.176,Z 763.396,A -85,B 0,C 180,E1 23007.908,E2 23007.908} C_VEL
LIN {X 0,Y 192.54,Z 737.455,A -85,B 0,C 180,E1 23014.182,E2 23014.182} C_VEL
LIN {X 0,Y 204.021,Z 719.765,A -85,B 0,C 180,E1 23017.144,E2 23017.144} C_VEL
LIN {X 0,Y 203.691,Z 704.6,A -85,B 0,C 180,E1 23024.357,E2 23024.357} C_VEL
LIN {X 0,Y 202.466,Z 694.321,A -85,B 0,C 180,E1 23031.42,E2 23031.42} C_VEL
LIN {X 0,Y 201.405,Z 688.619,A -85,B 0,C 180,E1 23037.845,E2 23037.845} C_VEL
LIN {X 0,Y 201.21,Z 687.379,A -85,B 0,C 180,E1 23039.992,E2 23039.992} C_VEL
LIN {X 0,Y 200.392,Z 686.978,A -85,B 0,C 180,E1 23044.31,E2 23044.31} C_VEL
LIN {X 0,Y 198.455,Z 691.728,A -85,B 0,C 180,E1 23053.176,E2 23053.176} C_VEL
LIN {X 0,Y 196.985,Z 699.663,A -85,B 0,C 180,E1 23060.551,E2 23060.551} C_VEL
LIN {X 0,Y 194.585,Z 710.443,A -85,B 0,C 180,E1 23067.717,E2 23067.717} C_VEL
LIN {X 0,Y 190.193,Z 723.808,A -85,B 0,C 180,E1 23075.052,E2 23075.052} C_VEL
LIN {X 0,Y 187.103,Z 728.646,A -85,B 0,C 180,E1 23076.996,E2 23076.996} C_VEL
LIN {X 0,Y 167.576,Z 749.344,A -85,B 0,C 180,E1 23084.845,E2 23084.845} C_VEL
LIN {X 0,Y 150.74,Z 764.233,A -85,B 0,C 180,E1 23094.866,E2 23094.866} C_VEL
LIN {X 0,Y 137.573,Z 774.643,A -85,B 0,C 180,E1 23108.458,E2 23108.458} C_VEL
LIN {X 0,Y 131.716,Z 779.158,A -85,B 0,C 180,E1 23123.427,E2 23123.427} C_VEL
LIN {X 0,Y 131.759,Z 779.122,A -85,B 0,C 180,E1 23136.582,E2 23136.582} C_VEL
LIN {X 0,Y 137.852,Z 774.406,A -85,B 0,C 180,E1 23151.844,E2 23151.844} C_VEL
LIN {X 0,Y 141.878,Z 771.231,A -85,B 0,C 180,E1 23157.062,E2 23157.062} C_VEL
LIN {X 0,Y 144.744,Z 766.963,A -85,B 0,C 180,E1 23163.773,E2 23163.773} C_VEL
LIN {X 0,Y 149.108,Z 761.56,A -85,B 0,C 180,E1 23170.064,E2 23170.064} C_VEL
LIN {X 0,Y 168.246,Z 744.669,A -85,B 0,C 180,E1 23179.676,E2 23179.676} C_VEL
LIN {X 0,Y 183.467,Z 728.385,A -85,B 0,C 180,E1 23185.337,E2 23185.337} C_VEL
LIN {X 0,Y 188.584,Z 715.791,A -85,B 0,C 180,E1 23192.567,E2 23192.567} C_VEL
LIN {X 0,Y 191.428,Z 706.085,A -85,B 0,C 180,E1 23199.237,E2 23199.237} C_VEL
LIN {X 0,Y 193.48,Z 698.345,A -85,B 0,C 180,E1 23206.478,E2 23206.478} C_VEL
LIN {X 0,Y 195.876,Z 693.404,A -85,B 0,C 180,E1 23215.59,E2 23215.59} C_VEL
LIN {X 0,Y 196.794,Z 693.801,A -85,B 0,C 180,E1 23220.008,E2 23220.008} C_VEL
LIN {X 0,Y 197.64,Z 699.775,A -85,B 0,C 180,E1 23227.728,E2 23227.728} C_VEL
LIN {X 0,Y 198.38,Z 710.27,A -85,B 0,C 180,E1 23235.179,E2 23235.179} C_VEL
LIN {X 0,Y 198.156,Z 722.314,A -85,B 0,C 180,E1 23241.256,E2 23241.256} C_VEL
LIN {X 0,Y 192.249,Z 731.572,A -85,B 0,C 180,E1 23242.878,E2 23242.878} C_VEL
LIN {X 0,Y 171.676,Z 757.761,A -85,B 0,C 180,E1 23248.477,E2 23248.477} C_VEL
LIN {X 0,Y 150.327,Z 780.731,A -85,B 0,C 180,E1 23257.177,E2 23257.177} C_VEL
LIN {X 0,Y 132.972,Z 798.287,A -85,B 0,C 180,E1 23269.263,E2 23269.263} C_VEL
LIN {X 0,Y 122.619,Z 810.338,A -85,B 0,C 180,E1 23284.481,E2 23284.481} C_VEL
LIN {X 0,Y 120.527,Z 815.289,A -85,B 0,C 180,E1 23295.493,E2 23295.493} C_VEL
LIN {X 0,Y 121.629,Z 818.031,A -85,B 0,C 180,E1 23309.994,E2 23309.994} C_VEL
LIN {X 0,Y 120.706,Z 817.219,A -85,B 0,C 180,E1 23317.175,E2 23317.175} C_VEL
LIN {X 0,Y 121.539,Z 812.297,A -85,B 0,C 180,E1 23331.86,E2 23331.86} C_VEL
LIN {X 0,Y 129.872,Z 801.499,A -85,B 0,C 180,E1 23347.58,E2 23347.58} C_VEL
LIN {X 0,Y 147.426,Z 783.809,A -85,B 0,C 180,E1 23361.291,E2 23361.291} C_VEL
LIN {X 0,Y 168.547,Z 761.495,A -85,B 0,C 180,E1 23370.457,E2 23370.457} C_VEL
LIN {X 0,Y 190.165,Z 734.831,A -85,B 0,C 180,E1 23376.617,E2 23376.617} C_VEL
LIN {X 0,Y 198.321,Z 722.414,A -85,B 0,C 180,E1 23378.751,E2 23378.751} C_VEL
LIN {X 0,Y 198.445,Z 708.336,A -85,B 0,C 180,E1 23386.091,E2 23386.091} C_VEL
LIN {X 0,Y 197.673,Z 699.386,A -85,B 0,C 180,E1 23392.874,E2 23392.874} C_VEL
LIN {X 0,Y 196.915,Z 694.061,A -85,B 0,C 180,E1 23399.992,E2 23399.992} C_VEL
LIN {X 0,Y 195.984,Z 693.701,A -85,B 0,C 180,E1 23404.407,E2 23404.407} C_VEL
LIN {X 0,Y 194.048,Z 697.273,A -85,B 0,C 180,E1 23411.798,E2 23411.798} C_VEL
LIN {X 0,Y 191.988,Z 704.663,A -85,B 0,C 180,E1 23419.427,E2 23419.427} C_VEL
LIN {X 0,Y 189.008,Z 715.091,A -85,B 0,C 180,E1 23426.805,E2 23426.805} C_VEL
LIN {X 0,Y 184.052,Z 727.575,A -85,B 0,C 180,E1 23434.056,E2 23434.056} C_VEL
LIN {X 0,Y 177.788,Z 735.067,A -85,B 0,C 180,E1 23436.629,E2 23436.629} C_VEL
LIN {X 0,Y 158.706,Z 753.624,A -85,B 0,C 180,E1 23444.521,E2 23444.521} C_VEL
LIN {X 0,Y 140.941,Z 768.105,A -85,B 0,C 180,E1 23455.807,E2 23455.807} C_VEL
LIN {X 0,Y 128.954,Z 776.813,A -85,B 0,C 180,E1 23469.455,E2 23469.455} C_VEL
LIN {X 0,Y 123.972,Z 780.342,A -85,B 0,C 180,E1 23483.015,E2 23483.015} C_VEL
LIN {X 0,Y 124.018,Z 780.306,A -85,B 0,C 180,E1 23496.994,E2 23496.994} C_VEL
LIN {X 0,Y 130.845,Z 775.44,A -85,B 0,C 180,E1 23513.45,E2 23513.45} C_VEL
LIN {X 0,Y 144.486,Z 765.249,A -85,B 0,C 180,E1 23526.911,E2 23526.911} C_VEL
LIN {X 0,Y 149.108,Z 761.56,A -85,B 0,C 180,E1 23530.064,E2 23530.064} C_VEL
LIN {X 0,Y 154.829,Z 755.127,A -85,B 0,C 180,E1 23535.816,E2 23535.816} C_VEL
LIN {X 0,Y 161.441,Z 747.534,A -85,B 0,C 180,E1 23541.038,E2 23541.038} C_VEL
LIN {X 0,Y 177.434,Z 731.628,A -85,B 0,C 180,E1 23546.74,E2 23546.74} C_VEL
LIN {X 0,Y 182.808,Z 720.629,A -85,B 0,C 180,E1 23553.333,E2 23553.333} C_VEL
LIN {X 0,Y 186.641,Z 710.112,A -85,B 0,C 180,E1 23561.142,E2 23561.142} C_VEL
LIN {X 0,Y 189.363,Z 702.781,A -85,B 0,C 180,E1 23569.28,E2 23569.28} C_VEL
LIN {X 0,Y 191.258,Z 700.032,A -85,B 0,C 180,E1 23575.484,E2 23575.484} C_VEL
LIN {X 0,Y 192.31,Z 700.369,A -85,B 0,C 180,E1 23580.008,E2 23580.008} C_VEL
LIN {X 0,Y 192.88,Z 706.548,A -85,B 0,C 180,E1 23587.92,E2 23587.92} C_VEL
LIN {X 0,Y 193.027,Z 717.012,A -85,B 0,C 180,E1 23595.305,E2 23595.305} C_VEL
LIN {X 0,Y 192.067,Z 726.401,A -85,B 0,C 180,E1 23600.027,E2 23600.027} C_VEL
LIN {X 0,Y 170.867,Z 753.088,A -85,B 0,C 180,E1 23605.144,E2 23605.144} C_VEL
LIN {X 0,Y 148.648,Z 776.461,A -85,B 0,C 180,E1 23613.119,E2 23613.119} C_VEL
LIN {X 0,Y 128.638,Z 795.306,A -85,B 0,C 180,E1 23625.259,E2 23625.259} C_VEL
LIN {X 0,Y 116.122,Z 807.999,A -85,B 0,C 180,E1 23640.831,E2 23640.831} C_VEL
LIN {X 0,Y 112.716,Z 814.06,A -85,B 0,C 180,E1 23654.464,E2 23654.464} C_VEL
LIN {X 0,Y 113.785,Z 816.84,A -85,B 0,C 180,E1 23669.994,E2 23669.994} C_VEL
LIN {X 0,Y 112.709,Z 814.089,A -85,B 0,C 180,E1 23685.524,E2 23685.524} C_VEL
LIN {X 0,Y 118.455,Z 805.407,A -85,B 0,C 180,E1 23703.405,E2 23703.405} C_VEL
LIN {X 0,Y 132.965,Z 791.341,A -85,B 0,C 180,E1 23718.099,E2 23718.099} C_VEL
LIN {X 0,Y 153.893,Z 771.459,A -85,B 0,C 180,E1 23729.076,E2 23729.076} C_VEL
LIN {X 0,Y 176.87,Z 746.275,A -85,B 0,C 180,E1 23736.496,E2 23736.496} C_VEL
LIN {X 0,Y 192.603,Z 725.981,A -85,B 0,C 180,E1 23740.06,E2 23740.06} C_VEL
LIN {X 0,Y 193.242,Z 714.312,A -85,B 0,C 180,E1 23746.444,E2 23746.444} C_VEL
LIN {X 0,Y 192.846,Z 704.734,A -85,B 0,C 180,E1 23754.101,E2 23754.101} C_VEL
LIN {X 0,Y 192.408,Z 700.639,A -85,B 0,C 180,E1 23759.992,E2 23759.992} C_VEL
LIN {X 0,Y 191.381,Z 700.279,A -85,B 0,C 180,E1 23764.513,E2 23764.513} C_VEL
LIN {X 0,Y 188.982,Z 704.256,A -85,B 0,C 180,E1 23772.509,E2 23772.509} C_VEL
LIN {X 0,Y 186.319,Z 711.68,A -85,B 0,C 180,E1 23780.043,E2 23780.043} C_VEL
LIN {X 0,Y 181.679,Z 723.589,A -85,B 0,C 180,E1 23788.36,E2 23788.36} C_VEL
LIN {X 0,Y 177.136,Z 732.215,A -85,B 0,C 180,E1 23793.298,E2 23793.298} C_VEL
LIN {X 0,Y 155.736,Z 752.767,A -85,B 0,C 180,E1 23801.339,E2 23801.339} C_VEL
LIN {X 0,Y 136.356,Z 768.04,A -85,B 0,C 180,E1 23812.516,E2 23812.516} C_VEL
LIN {X 0,Y 123.856,Z 776.574,A -85,B 0,C 180,E1 23824.767,E2 23824.767} C_VEL
LIN {X 0,Y 116.215,Z 781.53,A -85,B 0,C 180,E1 23842.546,E2 23842.546} C_VEL
LIN {X 0,Y 116.262,Z 781.494,A -85,B 0,C 180,E1 23857.464,E2 23857.464} C_VEL
LIN {X 0,Y 123.935,Z 776.462,A -85,B 0,C 180,E1 23875.228,E2 23875.228} C_VEL
LIN {X 0,Y 138.298,Z 766.447,A -85,B 0,C 180,E1 23888.862,E2 23888.862} C_VEL
LIN {X 0,Y 158.277,Z 750.439,A -85,B 0,C 180,E1 23899.707,E2 23899.707} C_VEL
LIN {X 0,Y 161.441,Z 747.534,A -85,B 0,C 180,E1 23901.038,E2 23901.038} C_VEL
LIN {X 0,Y 169.084,Z 738.815,A -85,B 0,C 180,E1 23905.641,E2 23905.641} C_VEL
LIN {X 0,Y 174.199,Z 730.565,A -85,B 0,C 180,E1 23910.676,E2 23910.676} C_VEL
LIN {X 0,Y 179.556,Z 719.596,A -85,B 0,C 180,E1 23918.365,E2 23918.365} C_VEL
LIN {X 0,Y 183.019,Z 711.773,A -85,B 0,C 180,E1 23925.69,E2 23925.69} C_VEL
LIN {X 0,Y 184.743,Z 708.352,A -85,B 0,C 180,E1 23930.608,E2 23930.608} C_VEL
LIN {X 0,Y 186.424,Z 706.505,A -85,B 0,C 180,E1 23935.366,E2 23935.366} C_VEL
LIN {X 0,Y 187.546,Z 706.742,A -85,B 0,C 180,E1 23940.009,E2 23940.009} C_VEL
LIN {X 0,Y 187.89,Z 713.145,A -85,B 0,C 180,E1 23948.087,E2 23948.087} C_VEL
LIN {X 0,Y 187.462,Z 722.822,A -85,B 0,C 180,E1 23954.99,E2 23954.99} C_VEL
LIN {X 0,Y 186.658,Z 728.764,A -85,B 0,C 180,E1 23958.257,E2 23958.257} C_VEL
LIN {X 0,Y 164.495,Z 755.169,A -85,B 0,C 180,E1 23963.454,E2 23963.454} C_VEL
LIN {X 0,Y 141.645,Z 777.6,A -85,B 0,C 180,E1 23971.536,E2 23971.536} C_VEL
LIN {X 0,Y 120.957,Z 795.765,A -85,B 0,C 180,E1 23984.159,E2 23984.159} C_VEL
LIN {X 0,Y 108.085,Z 807.852,A -85,B 0,C 180,E1 24000.743,E2 24000.743} C_VEL
LIN {X 0,Y 104.934,Z 812.83,A -85,B 0,C 180,E1 24013.279,E2 24013.279} C_VEL
LIN {X 0,Y 105.928,Z 815.646,A -85,B 0,C 180,E1 24029.993,E2 24029.993} C_VEL
LIN {X 0,Y 104.929,Z 812.859,A -85,B 0,C 180,E1 24046.707,E2 24046.707} C_VEL
LIN {X 0,Y 111.785,Z 804.042,A -85,B 0,C 180,E1 24065.892,E2 24065.892} C_VEL
LIN {X 0,Y 129.333,Z 788.623,A -85,B 0,C 180,E1 24081.945,E2 24081.945} C_VEL
LIN {X 0,Y 151.25,Z 768.829,A -85,B 0,C 180,E1 24092.29,E2 24092.29} C_VEL
LIN {X 0,Y 173.767,Z 744.978,A -85,B 0,C 180,E1 24098.973,E2 24098.973} C_VEL
LIN {X 0,Y 186.76,Z 728.94,A -85,B 0,C 180,E1 24101.745,E2 24101.745} C_VEL
LIN {X 0,Y 187.887,Z 717.915,A -85,B 0,C 180,E1 24108.279,E2 24108.279} C_VEL
LIN {X 0,Y 187.886,Z 710.029,A -85,B 0,C 180,E1 24115.385,E2 24115.385} C_VEL
LIN {X 0,Y 187.632,Z 707.024,A -85,B 0,C 180,E1 24119.991,E2 24119.991} C_VEL
LIN {X 0,Y 186.546,Z 706.745,A -85,B 0,C 180,E1 24124.631,E2 24124.631} C_VEL
LIN {X 0,Y 184.072,Z 710.048,A -85,B 0,C 180,E1 24131.814,E2 24131.814} C_VEL
LIN {X 0,Y 180.876,Z 717.228,A -85,B 0,C 180,E1 24139.483,E2 24139.483} C_VEL
LIN {X 0,Y 175.653,Z 728.246,A -85,B 0,C 180,E1 24147.593,E2 24147.593} C_VEL
LIN {X 0,Y 171.973,Z 734.514,A -85,B 0,C 180,E1 24151.451,E2 24151.451} C_VEL
LIN {X 0,Y 149.419,Z 754.996,A -85,B 0,C 180,E1 24159.652,E2 24159.652} C_VEL
LIN {X 0,Y 130.242,Z 769.23,A -85,B 0,C 180,E1 24170.424,E2 24170.424} C_VEL
LIN {X 0,Y 116.825,Z 777.763,A -85,B 0,C 180,E1 24183.131,E2 24183.131} C_VEL
LIN {X 0,Y 108.488,Z 782.714,A -85,B 0,C 180,E1 24202.012,E2 24202.012} C_VEL
LIN {X 0,Y 108.536,Z 782.679,A -85,B 0,C 180,E1 24217.998,E2 24217.998} C_VEL
LIN {X 0,Y 116.897,Z 777.654,A -85,B 0,C 180,E1 24236.865,E2 24236.865} C_VEL
LIN {X 0,Y 132.302,Z 767.639,A -85,B 0,C 180,E1 24250.987,E2 24250.987} C_VEL
LIN {X 0,Y 153.34,Z 751.647,A -85,B 0,C 180,E1 24261.935,E2 24261.935} C_VEL
LIN {X 0,Y 172.779,Z 733.058,A -85,B 0,C 180,E1 24269.12,E2 24269.12} C_VEL
LIN {X 0,Y 174.199,Z 730.565,A -85,B 0,C 180,E1 24270.676,E2 24270.676} C_VEL
LIN {X 0,Y 175.375,Z 726.388,A -85,B 0,C 180,E1 24274.72,E2 24274.72} C_VEL
LIN {X 0,Y 175.542,Z 721.526,A -85,B 0,C 180,E1 24281.894,E2 24281.894} C_VEL
LIN {X 0,Y 178.922,Z 715.481,A -85,B 0,C 180,E1 24288.947,E2 24288.947} C_VEL
LIN {X 0,Y 181.532,Z 712.67,A -85,B 0,C 180,E1 24295.966,E2 24295.966} C_VEL
LIN {X 0,Y 182.575,Z 712.975,A -85,B 0,C 180,E1 24300.009,E2 24300.009} C_VEL
LIN {X 0,Y 182.642,Z 718.73,A -85,B 0,C 180,E1 24307.494,E2 24307.494} C_VEL
LIN {X 0,Y 181.717,Z 728.038,A -85,B 0,C 180,E1 24314.433,E2 24314.433} C_VEL
LIN {X 0,Y 180.988,Z 731.705,A -85,B 0,C 180,E1 24316.465,E2 24316.465} C_VEL
LIN {X 0,Y 157.701,Z 757.633,A -85,B 0,C 180,E1 24321.798,E2 24321.798} C_VEL
LIN {X 0,Y 133.473,Z 779.803,A -85,B 0,C 180,E1 24330.371,E2 24330.371} C_VEL
LIN {X 0,Y 112.817,Z 796.548,A -85,B 0,C 180,E1 24343.378,E2 24343.378} C_VEL
LIN {X 0,Y 99.235,Z 808.521,A -85,B 0,C 180,E1 24362.852,E2 24362.852} C_VEL
LIN {X 0,Y 96.954,Z 813.558,A -85,B 0,C 180,E1 24381.039,E2 24381.039} C_VEL
LIN {X 0,Y 98.022,Z 814.445,A -85,B 0,C 180,E1 24389.993,E2 24389.993} C_VEL
LIN {X 0,Y 97.193,Z 811.628,A -85,B 0,C 180,E1 24408.081,E2 24408.081} C_VEL
LIN {X 0,Y 105.23,Z 802.789,A -85,B 0,C 180,E1 24428.519,E2 24428.519} C_VEL
LIN {X 0,Y 122.032,Z 789.284,A -85,B 0,C 180,E1 24443.477,E2 24443.477} C_VEL
LIN {X 0,Y 144.659,Z 770.216,A -85,B 0,C 180,E1 24454.102,E2 24454.102} C_VEL
LIN {X 0,Y 169.388,Z 745.519,A -85,B 0,C 180,E1 24461.157,E2 24461.157} C_VEL
LIN {X 0,Y 181.448,Z 731.097,A -85,B 0,C 180,E1 24463.822,E2 24463.822} C_VEL
LIN {X 0,Y 182.617,Z 721.29,A -85,B 0,C 180,E1 24470.479,E2 24470.479} C_VEL
LIN {X 0,Y 182.702,Z 714.614,A -85,B 0,C 180,E1 24477.625,E2 24477.625} C_VEL
LIN {X 0,Y 182.654,Z 713.24,A -85,B 0,C 180,E1 24479.991,E2 24479.991} C_VEL
LIN {X 0,Y 181.419,Z 713.019,A -85,B 0,C 180,E1 24484.762,E2 24484.762} C_VEL
LIN {X 0,Y 178.207,Z 717.077,A -85,B 0,C 180,E1 24492.986,E2 24492.986} C_VEL
LIN {X 0,Y 174.405,Z 724.192,A -85,B 0,C 180,E1 24500.237,E2 24500.237} C_VEL
LIN {X 0,Y 168.495,Z 734.432,A -85,B 0,C 180,E1 24507.964,E2 24507.964} C_VEL
LIN {X 0,Y 164.793,Z 738.813,A -85,B 0,C 180,E1 24510.123,E2 24510.123} C_VEL
LIN {X 0,Y 143.24,Z 757.226,A -85,B 0,C 180,E1 24517.817,E2 24517.817} C_VEL
LIN {X 0,Y 122.226,Z 771.677,A -85,B 0,C 180,E1 24529.607,E2 24529.607} C_VEL
LIN {X 0,Y 107.294,Z 780.378,A -85,B 0,C 180,E1 24545.053,E2 24545.053} C_VEL
LIN {X 0,Y 100.759,Z 783.9,A -85,B 0,C 180,E1 24561.395,E2 24561.395} C_VEL
LIN {X 0,Y 100.805,Z 783.865,A -85,B 0,C 180,E1 24578.616,E2 24578.616} C_VEL
LIN {X 0,Y 109.978,Z 778.845,A -85,B 0,C 180,E1 24598.706,E2 24598.706} C_VEL
LIN {X 0,Y 126.489,Z 768.836,A -85,B 0,C 180,E1 24613.317,E2 24613.317} C_VEL
LIN {X 0,Y 148.664,Z 752.85,A -85,B 0,C 180,E1 24624.299,E2 24624.299} C_VEL
LIN {X 0,Y 166.693,Z 736.714,A -85,B 0,C 180,E1 24630.455,E2 24630.455} C_VEL
LIN {X 0,Y 172.434,Z 727.377,A -85,B 0,C 180,E1 24636.915,E2 24636.915} C_VEL
LIN {X 0,Y 175.542,Z 721.526,A -85,B 0,C 180,E1 24641.894,E2 24641.894} C_VEL
LIN {X 0,Y 175.83,Z 719.615,A -85,B 0,C 180,E1 24646.115,E2 24646.115} C_VEL
LIN {X 0,Y 175.175,Z 719.56,A -85,B 0,C 180,E1 24653.474,E2 24653.474} C_VEL
LIN {X 0,Y 177.417,Z 719.061,A -85,B 0,C 180,E1 24660.009,E2 24660.009} C_VEL
LIN {X 0,Y 177.134,Z 725.041,A -85,B 0,C 180,E1 24667.728,E2 24667.728} C_VEL
LIN {X 0,Y 175.72,Z 733.773,A -85,B 0,C 180,E1 24674.275,E2 24674.275} C_VEL
LIN {X 0,Y 151.666,Z 759.414,A -85,B 0,C 180,E1 24679.818,E2 24679.818} C_VEL
LIN {X 0,Y 126.704,Z 780.737,A -85,B 0,C 180,E1 24688.461,E2 24688.461} C_VEL
LIN {X 0,Y 105.394,Z 796.703,A -85,B 0,C 180,E1 24701.85,E2 24701.85} C_VEL
LIN {X 0,Y 92.02,Z 807.274,A -85,B 0,C 180,E1 24720.523,E2 24720.523} C_VEL
LIN {X 0,Y 89.051,Z 812.341,A -85,B 0,C 180,E1 24740.236,E2 24740.236} C_VEL
LIN {X 0,Y 90.118,Z 813.244,A -85,B 0,C 180,E1 24749.992,E2 24749.992} C_VEL
LIN {X 0,Y 89.539,Z 810.401,A -85,B 0,C 180,E1 24769.688,E2 24769.688} C_VEL
LIN {X 0,Y 99.652,Z 800.976,A -85,B 0,C 180,E1 24792.352,E2 24792.352} C_VEL
LIN {X 0,Y 119.854,Z 786.099,A -85,B 0,C 180,E1 24808.179,E2 24808.179} C_VEL
LIN {X 0,Y 144.336,Z 766.276,A -85,B 0,C 180,E1 24818.082,E2 24818.082} C_VEL
LIN {X 0,Y 169.316,Z 741.631,A -85,B 0,C 180,E1 24824.28,E2 24824.28} C_VEL
LIN {X 0,Y 175.851,Z 733.911,A -85,B 0,C 180,E1 24825.729,E2 24825.729} C_VEL
LIN {X 0,Y 177.178,Z 725.523,A -85,B 0,C 180,E1 24832.044,E2 24832.044} C_VEL
LIN {X 0,Y 177.488,Z 719.312,A -85,B 0,C 180,E1 24839.991,E2 24839.991} C_VEL
LIN {X 0,Y 176.082,Z 719.146,A -85,B 0,C 180,E1 24844.907,E2 24844.907} C_VEL
LIN {X 0,Y 172.834,Z 722.691,A -85,B 0,C 180,E1 24852.465,E2 24852.465} C_VEL
LIN {X 0,Y 168.574,Z 729.264,A -85,B 0,C 180,E1 24859.569,E2 24859.569} C_VEL
LIN {X 0,Y 161.968,Z 739.06,A -85,B 0,C 180,E1 24867.308,E2 24867.308} C_VEL
LIN {X 0,Y 138.59,Z 758.423,A -85,B 0,C 180,E1 24875.266,E2 24875.266} C_VEL
LIN {X 0,Y 116.367,Z 772.868,A -85,B 0,C 180,E1 24887.105,E2 24887.105} C_VEL
LIN {X 0,Y 100.268,Z 781.565,A -85,B 0,C 180,E1 24903.17,E2 24903.17} C_VEL
LIN {X 0,Y 93.056,Z 785.084,A -85,B 0,C 180,E1 24920.676,E2 24920.676} C_VEL
LIN {X 0,Y 93.104,Z 785.05,A -85,B 0,C 180,E1 24939.335,E2 24939.335} C_VEL
LIN {X 0,Y 103.191,Z 780.035,A -85,B 0,C 180,E1 24960.791,E2 24960.791} C_VEL
LIN {X 0,Y 120.919,Z 770.031,A -85,B 0,C 180,E1 24975.859,E2 24975.859} C_VEL
LIN {X 0,Y 144.243,Z 754.056,A -85,B 0,C 180,E1 24986.821,E2 24986.821} C_VEL
LIN {X 0,Y 162.14,Z 738.56,A -85,B 0,C 180,E1 24992.866,E2 24992.866} C_VEL
LIN {X 0,Y 168.613,Z 728.862,A -85,B 0,C 180,E1 25000.558,E2 25000.558} C_VEL
LIN {X 0,Y 172.799,Z 722.372,A -85,B 0,C 180,E1 25007.677,E2 25007.677} C_VEL
LIN {X 0,Y 175.175,Z 719.56,A -85,B 0,C 180,E1 25013.474,E2 25013.474} C_VEL
LIN {X 0,Y 175.131,Z 720.382,A -85,B 0,C 180,E1 25017.017,E2 25017.017} C_VEL
LIN {X 0,Y 171.829,Z 728.185,A -85,B 0,C 180,E1 25024.824,E2 25024.824} C_VEL
LIN {X 0,Y 170.507,Z 735.51,A -85,B 0,C 180,E1 25031.476,E2 25031.476} C_VEL
LIN {X 0,Y 170.064,Z 737.128,A -85,B 0,C 180,E1 25032.561,E2 25032.561} C_VEL
LIN {X 0,Y 144.759,Z 761.988,A -85,B 0,C 180,E1 25037.965,E2 25037.965} C_VEL
LIN {X 0,Y 118.582,Z 782.722,A -85,B 0,C 180,E1 25047.021,E2 25047.021} C_VEL
LIN {X 0,Y 96.171,Z 798.06,A -85,B 0,C 180,E1 25061.806,E2 25061.806} C_VEL
LIN {X 0,Y 83.271,Z 807.548,A -85,B 0,C 180,E1 25082.521,E2 25082.521} C_VEL
LIN {X 0,Y 81.154,Z 811.121,A -85,B 0,C 180,E1 25099.275,E2 25099.275} C_VEL
LIN {X 0,Y 82.205,Z 812.042,A -85,B 0,C 180,E1 25109.991,E2 25109.991} C_VEL
LIN {X 0,Y 81.941,Z 809.168,A -85,B 0,C 180,E1 25131.601,E2 25131.601} C_VEL
LIN {X 0,Y 94.138,Z 799.464,A -85,B 0,C 180,E1 25156.15,E2 25156.15} C_VEL
LIN {X 0,Y 115.728,Z 784.844,A -85,B 0,C 180,E1 25171.641,E2 25171.641} C_VEL
LIN {X 0,Y 142.799,Z 763.871,A -85,B 0,C 180,E1 25181.507,E2 25181.507} C_VEL
LIN {X 0,Y 168.479,Z 739.103,A -85,B 0,C 180,E1 25187.159,E2 25187.159} C_VEL
LIN {X 0,Y 170.049,Z 737.43,A -85,B 0,C 180,E1 25187.422,E2 25187.422} C_VEL
LIN {X 0,Y 171.704,Z 729.752,A -85,B 0,C 180,E1 25193.684,E2 25193.684} C_VEL
LIN {X 0,Y 172.132,Z 725.238,A -85,B 0,C 180,E1 25199.991,E2 25199.991} C_VEL
LIN {X 0,Y 170.524,Z 725.141,A -85,B 0,C 180,E1 25205.067,E2 25205.067} C_VEL
LIN {X 0,Y 168.165,Z 727.203,A -85,B 0,C 180,E1 25210.328,E2 25210.328} C_VEL
LIN {X 0,Y 163.703,Z 732.948,A -85,B 0,C 180,E1 25217.583,E2 25217.583} C_VEL
LIN {X 0,Y 157.273,Z 741.249,A -85,B 0,C 180,E1 25224.822,E2 25224.822} C_VEL
LIN {X 0,Y 151.986,Z 746.027,A -85,B 0,C 180,E1 25226.692,E2 25226.692} C_VEL
LIN {X 0,Y 128.628,Z 763.37,A -85,B 0,C 180,E1 25234.809,E2 25234.809} C_VEL
LIN {X 0,Y 106.272,Z 776.48,A -85,B 0,C 180,E1 25247.599,E2 25247.599} C_VEL
LIN {X 0,Y 93.366,Z 782.75,A -85,B 0,C 180,E1 25261.007,E2 25261.007} C_VEL
LIN {X 0,Y 85.361,Z 786.27,A -85,B 0,C 180,E1 25279.827,E2 25279.827} C_VEL
LIN {X 0,Y 85.408,Z 786.236,A -85,B 0,C 180,E1 25300.185,E2 25300.185} C_VEL
LIN {X 0,Y 96.549,Z 781.226,A -85,B 0,C 180,E1 25323.17,E2 25323.17} C_VEL
LIN {X 0,Y 115.599,Z 771.228,A -85,B 0,C 180,E1 25338.647,E2 25338.647} C_VEL
LIN {X 0,Y 140.122,Z 755.259,A -85,B 0,C 180,E1 25349.494,E2 25349.494} C_VEL
LIN {X 0,Y 155.645,Z 742.704,A -85,B 0,C 180,E1 25354.247,E2 25354.247} C_VEL
LIN {X 0,Y 159.88,Z 737.72,A -85,B 0,C 180,E1 25357.832,E2 25357.832} C_VEL
LIN {X 0,Y 165.764,Z 729.774,A -85,B 0,C 180,E1 25365.659,E2 25365.659} C_VEL
LIN {X 0,Y 168.405,Z 726.599,A -85,B 0,C 180,E1 25370.292,E2 25370.292} C_VEL
LIN {X 0,Y 170.441,Z 724.911,A -85,B 0,C 180,E1 25374.931,E2 25374.931} C_VEL
LIN {X 0,Y 172.073,Z 724.989,A -85,B 0,C 180,E1 25380.009,E2 25380.009} C_VEL
LIN {X 0,Y 171.829,Z 728.185,A -85,B 0,C 180,E1 25384.824,E2 25384.824} C_VEL
LIN {X 0,Y 169.804,Z 732.786,A -85,B 0,C 180,E1 25387.988,E2 25387.988} C_VEL
LIN {X 0,Y 163.849,Z 740.633,A -85,B 0,C 180,E1 25390.548,E2 25390.548} C_VEL
LIN {X 0,Y 162.87,Z 741.683,A -85,B 0,C 180,E1 25390.749,E2 25390.749} C_VEL
LIN {X 0,Y 135.288,Z 766.599,A -85,B 0,C 180,E1 25396.632,E2 25396.632} C_VEL
LIN {X 0,Y 109.151,Z 785.375,A -85,B 0,C 180,E1 25406.014,E2 25406.014} C_VEL
LIN {X 0,Y 86.57,Z 799.46,A -85,B 0,C 180,E1 25422.19,E2 25422.19} C_VEL
LIN {X 0,Y 74.422,Z 807.897,A -85,B 0,C 180,E1 25446.067,E2 25446.067} C_VEL
LIN {X 0,Y 74.285,Z 810.839,A -85,B 0,C 180,E1 25469.99,E2 25469.99} C_VEL
LIN {X 0,Y 74.458,Z 807.936,A -85,B 0,C 180,E1 25493.9,E2 25493.9} C_VEL
LIN {X 0,Y 88.634,Z 798.212,A -85,B 0,C 180,E1 25519.991,E2 25519.991} C_VEL
LIN {X 0,Y 112.062,Z 783.591,A -85,B 0,C 180,E1 25535.336,E2 25535.336} C_VEL
LIN {X 0,Y 139.56,Z 763.322,A -85,B 0,C 180,E1 25544.468,E2 25544.468} C_VEL
LIN {X 0,Y 163.728,Z 741.068,A -85,B 0,C 180,E1 25549.369,E2 25549.369} C_VEL
LIN {X 0,Y 165.161,Z 738.504,A -85,B 0,C 180,E1 25550.792,E2 25550.792} C_VEL
LIN {X 0,Y 166.416,Z 731.927,A -85,B 0,C 180,E1 25558.267,E2 25558.267} C_VEL
LIN {X 0,Y 166.014,Z 730.87,A -85,B 0,C 180,E1 25561.352,E2 25561.352} C_VEL
LIN {X 0,Y 164.023,Z 731.421,A -85,B 0,C 180,E1 25566.652,E2 25566.652} C_VEL
LIN {X 0,Y 160.189,Z 735.118,A -85,B 0,C 180,E1 25573.61,E2 25573.61} C_VEL
LIN {X 0,Y 154.076,Z 742.051,A -85,B 0,C 180,E1 25580.9,E2 25580.9} C_VEL
LIN {X 0,Y 151.233,Z 745.173,A -85,B 0,C 180,E1 25583.342,E2 25583.342} C_VEL
LIN {X 0,Y 127.231,Z 762.728,A -85,B 0,C 180,E1 25590.714,E2 25590.714} C_VEL
LIN {X 0,Y 103.013,Z 776.489,A -85,B 0,C 180,E1 25602.923,E2 25602.923} C_VEL
LIN {X 0,Y 86.592,Z 783.939,A -85,B 0,C 180,E1 25618.492,E2 25618.492} C_VEL
LIN {X 0,Y 77.696,Z 787.454,A -85,B 0,C 180,E1 25638.811,E2 25638.811} C_VEL
LIN {X 0,Y 77.746,Z 787.421,A -85,B 0,C 180,E1 25661.201,E2 25661.201} C_VEL
LIN {X 0,Y 90.109,Z 782.416,A -85,B 0,C 180,E1 25685.89,E2 25685.89} C_VEL
LIN {X 0,Y 110.558,Z 772.437,A -85,B 0,C 180,E1 25701.684,E2 25701.684} C_VEL
LIN {X 0,Y 136.315,Z 756.465,A -85,B 0,C 180,E1 25712.33,E2 25712.33} C_VEL
LIN {X 0,Y 151.269,Z 744.906,A -85,B 0,C 180,E1 25716.641,E2 25716.641} C_VEL
LIN {X 0,Y 157.808,Z 737.466,A -85,B 0,C 180,E1 25723.342,E2 25723.342} C_VEL
LIN {X 0,Y 161.875,Z 732.95,A -85,B 0,C 180,E1 25729.266,E2 25729.266} C_VEL
LIN {X 0,Y 164.769,Z 730.739,A -85,B 0,C 180,E1 25735.089,E2 25735.089} C_VEL
LIN {X 0,Y 166.472,Z 730.691,A -85,B 0,C 180,E1 25740.01,E2 25740.01} C_VEL
LIN {X 0,Y 165.487,Z 736.747,A -85,B 0,C 180,E1 25747.785,E2 25747.785} C_VEL
LIN {X 0,Y 164.818,Z 739.148,A -85,B 0,C 180,E1 25749.872,E2 25749.872} C_VEL
LIN {X 0,Y 162.87,Z 741.683,A -85,B 0,C 180,E1 25750.749,E2 25750.749} C_VEL
LIN {X 0,Y 156.609,Z 747.535,A -85,B 0,C 180,E1 25751.391,E2 25751.391} C_VEL
LIN {X 0,Y 137.384,Z 762.087,A -85,B 0,C 180,E1 25752.323,E2 25752.323} C_VEL
LIN {X 0,Y 135.755,Z 763.341,A -85,B 0,C 180,E1 25752.644,E2 25752.644} C_VEL
LIN {X 0,Y 108.916,Z 782.207,A -85,B 0,C 180,E1 25760.731,E2 25760.731} C_VEL
LIN {X 0,Y 83.635,Z 796.886,A -85,B 0,C 180,E1 25775.706,E2 25775.706} C_VEL
LIN {X 0,Y 67.048,Z 806.658,A -85,B 0,C 180,E1 25803.238,E2 25803.238} C_VEL
LIN {X 0,Y 66.351,Z 809.634,A -85,B 0,C 180,E1 25829.989,E2 25829.989} C_VEL
LIN {X 0,Y 67.102,Z 806.702,A -85,B 0,C 180,E1 25856.715,E2 25856.715} C_VEL
LIN {X 0,Y 83.6,Z 796.964,A -85,B 0,C 180,E1 25884.298,E2 25884.298} C_VEL
LIN {X 0,Y 108.888,Z 782.336,A -85,B 0,C 180,E1 25899.271,E2 25899.271} C_VEL
LIN {X 0,Y 137.443,Z 762.166,A -85,B 0,C 180,E1 25907.733,E2 25907.733} C_VEL
LIN {X 0,Y 158.757,Z 743.459,A -85,B 0,C 180,E1 25911.665,E2 25911.665} C_VEL
LIN {X 0,Y 160.337,Z 738.705,A -85,B 0,C 180,E1 25916.41,E2 25916.41} C_VEL
LIN {X 0,Y 160.734,Z 736.461,A -85,B 0,C 180,E1 25919.99,E2 25919.99} C_VEL
LIN {X 0,Y 158.762,Z 736.559,A -85,B 0,C 180,E1 25925.443,E2 25925.443} C_VEL
LIN {X 0,Y 154.558,Z 739.838,A -85,B 0,C 180,E1 25932.526,E2 25932.526} C_VEL
LIN {X 0,Y 147.606,Z 746.788,A -85,B 0,C 180,E1 25940.188,E2 25940.188} C_VEL
LIN {X 0,Y 141.994,Z 751.286,A -85,B 0,C 180,E1 25942.106,E2 25942.106} C_VEL
LIN {X 0,Y 114.449,Z 769.184,A -85,B 0,C 180,E1 25951.034,E2 25951.034} C_VEL
LIN {X 0,Y 90.418,Z 780.995,A -85,B 0,C 180,E1 25964.837,E2 25964.837} C_VEL
LIN {X 0,Y 73.836,Z 787.373,A -85,B 0,C 180,E1 25985.886,E2 25985.886} C_VEL
LIN {X 0,Y 68.372,Z 789.168,A -85,B 0,C 180,E1 26010.011,E2 26010.011} C_VEL
LIN {X 0,Y 73.929,Z 787.317,A -85,B 0,C 180,E1 26034.103,E2 26034.103} C_VEL
LIN {X 0,Y 92.86,Z 779.816,A -85,B 0,C 180,E1 26057,E2 26057} C_VEL
LIN {X 0,Y 117.472,Z 767.374,A -85,B 0,C 180,E1 26070.128,E2 26070.128} C_VEL
LIN {X 0,Y 144.768,Z 748.914,A -85,B 0,C 180,E1 26078.522,E2 26078.522} C_VEL
LIN {X 0,Y 148.576,Z 745.561,A -85,B 0,C 180,E1 26080.737,E2 26080.737} C_VEL
LIN {X 0,Y 154.544,Z 739.576,A -85,B 0,C 180,E1 26087.54,E2 26087.54} C_VEL
LIN {X 0,Y 158.682,Z 736.349,A -85,B 0,C 180,E1 26094.554,E2 26094.554} C_VEL
LIN {X 0,Y 160.68,Z 736.237,A -85,B 0,C 180,E1 26100.01,E2 26100.01} C_VEL
LIN {X 0,Y 159.512,Z 741.629,A -85,B 0,C 180,E1 26107.155,E2 26107.155} C_VEL
LIN {X 0,Y 158.701,Z 743.265,A -85,B 0,C 180,E1 26108.333,E2 26108.333} C_VEL
LIN {X 0,Y 135.755,Z 763.341,A -85,B 0,C 180,E1 26112.644,E2 26112.644} C_VEL
LIN {X 0,Y 121.277,Z 772.661,A -85,B 0,C 180,E1 26114.22,E2 26114.22} C_VEL
LIN {X 0,Y 108.154,Z 779.871,A -85,B 0,C 180,E1 26115.969,E2 26115.969} C_VEL
LIN {X 0,Y 106.464,Z 780.838,A -85,B 0,C 180,E1 26116.504,E2 26116.504} C_VEL
LIN {X 0,Y 79.107,Z 795.63,A -85,B 0,C 180,E1 26130.85,E2 26130.85} C_VEL
LIN {X 0,Y 62.294,Z 803.964,A -85,B 0,C 180,E1 26152.716,E2 26152.716} C_VEL
LIN {X 0,Y 57.598,Z 807.451,A -85,B 0,C 180,E1 26174.8,E2 26174.8} C_VEL
LIN {X 0,Y 58.425,Z 808.43,A -85,B 0,C 180,E1 26189.988,E2 26189.988} C_VEL
LIN {X 0,Y 59.923,Z 805.463,A -85,B 0,C 180,E1 26220.225,E2 26220.225} C_VEL
LIN {X 0,Y 79.076,Z 795.712,A -85,B 0,C 180,E1 26249.151,E2 26249.151} C_VEL
LIN {X 0,Y 106.605,Z 780.882,A -85,B 0,C 180,E1 26263.54,E2 26263.54} C_VEL
LIN {X 0,Y 135.936,Z 760.891,A -85,B 0,C 180,E1 26271.117,E2 26271.117} C_VEL
LIN {X 0,Y 153.69,Z 745.726,A -85,B 0,C 180,E1 26274.355,E2 26274.355} C_VEL
LIN {X 0,Y 154.786,Z 741.8,A -85,B 0,C 180,E1 26279.99,E2 26279.99} C_VEL
LIN {X 0,Y 151.895,Z 742.348,A -85,B 0,C 180,E1 26286.632,E2 26286.632} C_VEL
LIN {X 0,Y 147.456,Z 745.66,A -85,B 0,C 180,E1 26293.14,E2 26293.14} C_VEL
LIN {X 0,Y 141.153,Z 751.049,A -85,B 0,C 180,E1 26298.692,E2 26298.692} C_VEL
LIN {X 0,Y 113.707,Z 768.747,A -85,B 0,C 180,E1 26306.411,E2 26306.411} C_VEL
LIN {X 0,Y 87.667,Z 781.112,A -85,B 0,C 180,E1 26319.25,E2 26319.25} C_VEL
LIN {X 0,Y 69.97,Z 787.534,A -85,B 0,C 180,E1 26337.388,E2 26337.388} C_VEL
LIN {X 0,Y 62.451,Z 789.825,A -85,B 0,C 180,E1 26356.03,E2 26356.03} C_VEL
LIN {X 0,Y 63.733,Z 789.472,A -85,B 0,C 180,E1 26388.82,E2 26388.82} C_VEL
LIN {X 0,Y 77.992,Z 784.793,A -85,B 0,C 180,E1 26412.634,E2 26412.634} C_VEL
LIN {X 0,Y 101.571,Z 774.846,A -85,B 0,C 180,E1 26428.584,E2 26428.584} C_VEL
LIN {X 0,Y 129.797,Z 758.87,A -85,B 0,C 180,E1 26438.453,E2 26438.453} C_VEL
LIN {X 0,Y 141.715,Z 750.409,A -85,B 0,C 180,E1 26441.385,E2 26441.385} C_VEL
LIN {X 0,Y 148.589,Z 744.477,A -85,B 0,C 180,E1 26448.293,E2 26448.293} C_VEL
LIN {X 0,Y 152.807,Z 741.745,A -85,B 0,C 180,E1 26455.551,E2 26455.551} C_VEL
LIN {X 0,Y 154.733,Z 741.597,A -85,B 0,C 180,E1 26460.01,E2 26460.01} C_VEL
LIN {X 0,Y 153.645,Z 745.528,A -85,B 0,C 180,E1 26465.646,E2 26465.646} C_VEL
LIN {X 0,Y 127.478,Z 767.032,A -85,B 0,C 180,E1 26470.656,E2 26470.656} C_VEL
LIN {X 0,Y 106.464,Z 780.838,A -85,B 0,C 180,E1 26476.504,E2 26476.504} C_VEL
LIN {X 0,Y 91.449,Z 787.933,A -85,B 0,C 180,E1 26479.831,E2 26479.831} C_VEL
LIN {X 0,Y 76.488,Z 793.804,A -85,B 0,C 180,E1 26484.604,E2 26484.604} C_VEL
LIN {X 0,Y 56.007,Z 802.721,A -85,B 0,C 180,E1 26507.641,E2 26507.641} C_VEL
LIN {X 0,Y 49.871,Z 806.228,A -85,B 0,C 180,E1 26532.373,E2 26532.373} C_VEL
LIN {X 0,Y 50.468,Z 807.221,A -85,B 0,C 180,E1 26549.986,E2 26549.986} C_VEL
LIN {X 0,Y 53.014,Z 804.22,A -85,B 0,C 180,E1 26584.681,E2 26584.681} C_VEL
LIN {X 0,Y 74.968,Z 794.562,A -85,B 0,C 180,E1 26614.387,E2 26614.387} C_VEL
LIN {X 0,Y 105.663,Z 779.015,A -85,B 0,C 180,E1 26628.211,E2 26628.211} C_VEL
LIN {X 0,Y 136.356,Z 758.52,A -85,B 0,C 180,E1 26634.778,E2 26634.778} C_VEL
LIN {X 0,Y 146.286,Z 750.555,A -85,B 0,C 180,E1 26636.219,E2 26636.219} C_VEL
LIN {X 0,Y 148.102,Z 748.732,A -85,B 0,C 180,E1 26637.069,E2 26637.069} C_VEL
LIN {X 0,Y 148.645,Z 746.983,A -85,B 0,C 180,E1 26639.989,E2 26639.989} C_VEL
LIN {X 0,Y 146,Z 747.286,A -85,B 0,C 180,E1 26645.921,E2 26645.921} C_VEL
LIN {X 0,Y 141.251,Z 750.383,A -85,B 0,C 180,E1 26652.324,E2 26652.324} C_VEL
LIN {X 0,Y 136.458,Z 754.018,A -85,B 0,C 180,E1 26656.119,E2 26656.119} C_VEL
LIN {X 0,Y 107.226,Z 771.573,A -85,B 0,C 180,E1 26663.853,E2 26663.853} C_VEL
LIN {X 0,Y 82.932,Z 782.304,A -85,B 0,C 180,E1 26675.055,E2 26675.055} C_VEL
LIN {X 0,Y 63.538,Z 788.719,A -85,B 0,C 180,E1 26693.594,E2 26693.594} C_VEL
LIN {X 0,Y 54.914,Z 791.01,A -85,B 0,C 180,E1 26714.065,E2 26714.065} C_VEL
LIN {X 0,Y 54.97,Z 790.979,A -85,B 0,C 180,E1 26745.946,E2 26745.946} C_VEL
LIN {X 0,Y 72.424,Z 785.985,A -85,B 0,C 180,E1 26776.835,E2 26776.835} C_VEL
LIN {X 0,Y 97.029,Z 776.363,A -85,B 0,C 180,E1 26792.21,E2 26792.21} C_VEL
LIN {X 0,Y 125.449,Z 761.103,A -85,B 0,C 180,E1 26801.319,E2 26801.319} C_VEL
LIN {X 0,Y 137.269,Z 753.207,A -85,B 0,C 180,E1 26803.976,E2 26803.976} C_VEL
LIN {X 0,Y 143.869,Z 748.29,A -85,B 0,C 180,E1 26810.96,E2 26810.96} C_VEL
LIN {X 0,Y 146.651,Z 746.945,A -85,B 0,C 180,E1 26815.886,E2 26815.886} C_VEL
LIN {X 0,Y 148.591,Z 746.791,A -85,B 0,C 180,E1 26820.011,E2 26820.011} C_VEL
LIN {X 0,Y 148.096,Z 748.517,A -85,B 0,C 180,E1 26822.931,E2 26822.931} C_VEL
LIN {X 0,Y 143.733,Z 752.462,A -85,B 0,C 180,E1 26824.13,E2 26824.13} C_VEL
LIN {X 0,Y 112.969,Z 774.499,A -85,B 0,C 180,E1 26829.876,E2 26829.876} C_VEL
LIN {X 0,Y 84.326,Z 790.124,A -85,B 0,C 180,E1 26840.019,E2 26840.019} C_VEL
LIN {X 0,Y 76.488,Z 793.804,A -85,B 0,C 180,E1 26844.604,E2 26844.604} C_VEL
LIN {X 0,Y 62.058,Z 798.549,A -85,B 0,C 180,E1 26851.949,E2 26851.949} C_VEL
LIN {X 0,Y 49.027,Z 801.918,A -85,B 0,C 180,E1 26863.68,E2 26863.68} C_VEL
LIN {X 0,Y 42.253,Z 805.002,A -85,B 0,C 180,E1 26889.058,E2 26889.058} C_VEL
LIN {X 0,Y 42.507,Z 806.012,A -85,B 0,C 180,E1 26909.983,E2 26909.983} C_VEL
LIN {X 0,Y 46.526,Z 802.98,A -85,B 0,C 180,E1 26950.418,E2 26950.418} C_VEL
LIN {X 0,Y 71.422,Z 793.473,A -85,B 0,C 180,E1 26980.076,E2 26980.076} C_VEL
LIN {X 0,Y 104.249,Z 777.786,A -85,B 0,C 180,E1 26992.622,E2 26992.622} C_VEL
LIN {X 0,Y 135.854,Z 757.249,A -85,B 0,C 180,E1 26998.232,E2 26998.232} C_VEL
LIN {X 0,Y 142.098,Z 752.323,A -85,B 0,C 180,E1 26999.292,E2 26999.292} C_VEL
LIN {X 0,Y 139.184,Z 752.458,A -85,B 0,C 180,E1 27006.212,E2 27006.212} C_VEL
LIN {X 0,Y 134.915,Z 754.946,A -85,B 0,C 180,E1 27011.432,E2 27011.432} C_VEL
LIN {X 0,Y 132.941,Z 756.258,A -85,B 0,C 180,E1 27013.108,E2 27013.108} C_VEL
LIN {X 0,Y 104.304,Z 772.77,A -85,B 0,C 180,E1 27019.915,E2 27019.915} C_VEL
LIN {X 0,Y 78.703,Z 783.493,A -85,B 0,C 180,E1 27030.391,E2 27030.391} C_VEL
LIN {X 0,Y 57.425,Z 789.908,A -85,B 0,C 180,E1 27048.952,E2 27048.952} C_VEL
LIN {X 0,Y 47.469,Z 792.193,A -85,B 0,C 180,E1 27071.482,E2 27071.482} C_VEL
LIN {X 0,Y 47.526,Z 792.162,A -85,B 0,C 180,E1 27108.528,E2 27108.528} C_VEL
LIN {X 0,Y 67.309,Z 787.176,A -85,B 0,C 180,E1 27141.703,E2 27141.703} C_VEL
LIN {X 0,Y 95.292,Z 776.821,A -85,B 0,C 180,E1 27157.069,E2 27157.069} C_VEL
LIN {X 0,Y 124.908,Z 761.271,A -85,B 0,C 180,E1 27165.133,E2 27165.133} C_VEL
LIN {X 0,Y 132.983,Z 756.031,A -85,B 0,C 180,E1 27166.896,E2 27166.896} C_VEL
LIN {X 0,Y 139.249,Z 752.201,A -85,B 0,C 180,E1 27173.791,E2 27173.791} C_VEL
LIN {X 0,Y 142.069,Z 752.127,A -85,B 0,C 180,E1 27180.721,E2 27180.721} C_VEL
LIN {X 0,Y 111.856,Z 773.244,A -85,B 0,C 180,E1 27185.739,E2 27185.739} C_VEL
LIN {X 0,Y 81.878,Z 788.872,A -85,B 0,C 180,E1 27194.608,E2 27194.608} C_VEL
LIN {X 0,Y 54.841,Z 799.794,A -85,B 0,C 180,E1 27214.344,E2 27214.344} C_VEL
LIN {X 0,Y 49.027,Z 801.918,A -85,B 0,C 180,E1 27223.68,E2 27223.68} C_VEL
LIN {X 0,Y 41.448,Z 803.74,A -85,B 0,C 180,E1 27237.166,E2 27237.166} C_VEL
LIN {X 0,Y 34.18,Z 804.678,A -85,B 0,C 180,E1 27265.688,E2 27265.688} C_VEL
LIN {X 0,Y 34.452,Z 804.774,A -85,B 0,C 180,E1 27269.345,E2 27269.345} C_VEL
LIN {X 0,Y 36.066,Z 803.299,A -85,B 0,C 180,E1 27303.122,E2 27303.122} C_VEL
LIN {X 0,Y 59.778,Z 795.582,A -85,B 0,C 180,E1 27341.15,E2 27341.15} C_VEL
LIN {X 0,Y 90.968,Z 782.853,A -85,B 0,C 180,E1 27354.325,E2 27354.325} C_VEL
